SPLINE
SPL {X  -162.485, Y  +370.062, Z    +0.000, E1   +10.606, E3 +501495.136}
SPL {X  -162.818, Y  +379.636, Z    +0.000, E1    +5.115, E3 +501484.485}
SPL {X  -162.820, Y  +386.976, Z    +0.000, E1    +0.144, E3 +501483.584}
SPL {X  -162.820, Y  +390.236, Z    +0.000, E1    -2.204, E3 +501489.642}
SPL {X  -162.820, Y  +393.415, Z    +0.000, E1    -4.587, E3 +501490.927}
SPL {X  -162.820, Y  +399.630, Z    +0.000, E1    -9.426, E3 +501492.856}
SPL {X  -162.820, Y  +408.127, Z    +0.000, E1   -18.417, E3 +501479.144}
SPL {X  -162.820, Y  +420.083, Z    +0.000, E1   -24.325, E3 +501499.620}
SPL {X  -162.820, Y  +428.527, Z    +0.000, E1   -26.988, E3 +501516.912}
SPL {X  -162.820, Y  +431.336, Z    +0.000, E1   -24.162, E3 +501547.122}
SPL {X  -162.820, Y  +432.048, Z    +0.000, E1   -22.832, E3 +501561.626}
SPL {X  -162.820, Y  +434.888, Z    +0.000, E1   -22.823, E3 +501575.575}
SPL {X  -162.820, Y  +436.834, Z    +0.000, E1   -22.779, E3 +501585.535}
SPL {X  -162.820, Y  +438.868, Z    +0.000, E1   -22.837, E3 +501595.189}
SPL {X  -162.820, Y  +441.351, Z    +0.000, E1   -22.805, E3 +501607.764}
SPL {X  -162.820, Y  +443.809, Z    +0.000, E1   -22.804, E3 +501619.930}
SPL {X  -162.820, Y  +447.077, Z    +0.000, E1   -22.869, E3 +501635.741}
SPL {X  -162.820, Y  +449.911, Z    +0.000, E1   -22.774, E3 +501650.350}
SPL {X  -162.820, Y  +451.861, Z    +0.000, E1   -22.750, E3 +501660.198}
SPL {X  -162.820, Y  +454.167, Z    +0.000, E1   -22.842, E3 +501670.927}
SPL {X  -162.820, Y  +456.529, Z    +0.000, E1   -22.855, E3 +501682.456}
SPL {X  -162.820, Y  +458.725, Z    +0.000, E1   -22.793, E3 +501693.860}
SPL {X  -162.820, Y  +460.754, Z    +0.000, E1   -22.806, E3 +501703.733}
SPL {X  -162.820, Y  +462.409, Z    +0.000, E1   -22.783, E3 +501712.150}
SPL {X  -162.820, Y  +464.633, Z    +0.000, E1   -22.813, E3 +501722.979}
SPL {X  -162.820, Y  +467.913, Z    +0.000, E1   -22.879, E3 +501738.819}
SPL {X  -162.820, Y  +470.892, Z    +0.000, E1   -22.837, E3 +501753.708}
SPL {X  -162.820, Y  +472.726, Z    +0.000, E1   -22.777, E3 +501763.247}
SPL {X  -162.820, Y  +475.118, Z    +0.000, E1   -22.777, E3 +501775.218}
SPL {X  -162.820, Y  +477.389, Z    +0.000, E1   -22.803, E3 +501786.135}
SPL {X  -162.820, Y  +478.914, Z    +0.000, E1   -22.821, E3 +501793.526}
SPL {X  -162.820, Y  +481.034, Z    +0.000, E1   -22.831, E3 +501804.048}
SPL {X  -162.820, Y  +484.256, Z    +0.000, E1   -22.840, E3 +501820.067}
SPL {X  -162.820, Y  +487.952, Z    +0.000, E1   -22.824, E3 +501838.497}
SPL {X  -162.820, Y  +491.768, Z    +0.000, E1   -22.852, E3 +501857.178}
SPL {X  -162.820, Y  +495.526, Z    +0.000, E1   -22.833, E3 +501875.949}
SPL {X  -162.820, Y  +499.330, Z    +0.000, E1   -22.841, E3 +501894.730}
SPL {X  -162.820, Y  +503.049, Z    +0.000, E1   -22.823, E3 +501913.280}
SPL {X  -162.820, Y  +506.908, Z    +0.000, E1   -22.877, E3 +501931.950}
SPL {X  -162.820, Y  +510.068, Z    +0.000, E1   -22.761, E3 +501948.421}
SPL {X  -162.820, Y  +512.359, Z    +0.000, E1   -22.823, E3 +501959.153}
SPL {X  -162.820, Y  +514.562, Z    +0.000, E1   -22.806, E3 +501970.340}
SPL {X  -162.820, Y  +517.952, Z    +0.000, E1   -22.864, E3 +501986.737}
SPL {X  -162.820, Y  +520.641, Z    +0.000, E1   -22.790, E3 +502000.456}
SPL {X  -162.820, Y  +522.740, Z    +0.000, E1   -22.811, E3 +502010.698}
SPL {X  -162.820, Y  +524.628, Z    +0.000, E1   -22.846, E3 +502019.693}
SPL {X  -162.820, Y  +526.661, Z    +0.000, E1   -22.801, E3 +502030.249}
SPL {X  -162.820, Y  +529.662, Z    +0.000, E1   -22.810, E3 +502045.099}
SPL {X  -162.820, Y  +532.614, Z    +0.000, E1   -22.828, E3 +502059.506}
SPL {X  -162.820, Y  +534.838, Z    +0.000, E1   -22.864, E3 +502070.134}
SPL {X  -162.820, Y  +536.882, Z    +0.000, E1   -22.782, E3 +502080.989}
SPL {X  -162.820, Y  +539.194, Z    +0.000, E1   -22.826, E3 +502092.038}
SPL {X  -162.820, Y  +541.555, Z    +0.000, E1   -22.817, E3 +502103.852}
SPL {X  -162.820, Y  +543.728, Z    +0.000, E1   -22.799, E3 +502114.710}
SPL {X  -162.820, Y  +545.925, Z    +0.000, E1   -22.803, E3 +502125.580}
SPL {X  -162.820, Y  +548.328, Z    +0.000, E1   -22.796, E3 +502137.575}
SPL {X  -162.820, Y  +551.027, Z    +0.000, E1   -22.819, E3 +502150.768}
SPL {X  -162.820, Y  +553.721, Z    +0.000, E1   -22.807, E3 +502164.212}
SPL {X  -162.820, Y  +556.430, Z    +0.000, E1   -22.821, E3 +502177.508}
SPL {X  -162.820, Y  +558.974, Z    +0.000, E1   -22.806, E3 +502190.208}
SPL {X  -162.820, Y  +562.171, Z    +0.000, E1   -22.845, E3 +502205.906}
SPL {X  -162.820, Y  +565.170, Z    +0.000, E1   -22.801, E3 +502220.919}
SPL {X  -162.820, Y  +567.308, Z    +0.000, E1   -22.750, E3 +502231.936}
SPL {X  -162.820, Y  +570.378, Z    +0.000, E1   -22.843, E3 +502246.559}
SPL {X  -162.820, Y  +573.634, Z    +0.000, E1   -22.827, E3 +502262.703}
SPL {X  -162.820, Y  +576.228, Z    +0.000, E1   -22.814, E3 +502275.600}
SPL {X  -162.820, Y  +578.553, Z    +0.000, E1   -22.801, E3 +502287.215}
SPL {X  -162.820, Y  +581.064, Z    +0.000, E1   -22.823, E3 +502299.500}
SPL {X  -162.820, Y  +583.435, Z    +0.000, E1   -22.808, E3 +502311.322}
SPL {X  -162.820, Y  +585.410, Z    +0.000, E1   -22.764, E3 +502321.457}
SPL {X  -162.820, Y  +587.676, Z    +0.000, E1   -22.853, E3 +502331.972}
SPL {X  -162.820, Y  +590.707, Z    +0.000, E1   -22.855, E3 +502347.122}
SPL {X  -162.820, Y  +593.650, Z    +0.000, E1   -22.810, E3 +502361.882}
SPL {X  -162.820, Y  +595.830, Z    +0.000, E1   -22.828, E3 +502372.498}
SPL {X  -162.820, Y  +598.094, Z    +0.000, E1   -22.843, E3 +502383.611}
SPL {X  -162.820, Y  +600.420, Z    +0.000, E1   -22.826, E3 +502395.243}
SPL {X  -162.820, Y  +602.573, Z    +0.000, E1   -22.830, E3 +502405.828}
SPL {X  -162.820, Y  +604.828, Z    +0.000, E1   -22.784, E3 +502417.466}
SPL {X  -162.820, Y  +607.142, Z    +0.000, E1   -22.808, E3 +502428.647}
SPL {X  -162.820, Y  +608.890, Z    +0.000, E1   -22.790, E3 +502437.471}
SPL {X  -162.820, Y  +611.103, Z    +0.000, E1   -22.785, E3 +502448.510}
SPL {X  -162.820, Y  +613.294, Z    +0.000, E1   -22.780, E3 +502459.383}
SPL {X  -162.820, Y  +615.356, Z    +0.000, E1   -22.799, E3 +502469.440}
SPL {X  -162.820, Y  +617.439, Z    +0.000, E1   -22.808, E3 +502479.698}
SPL {X  -162.820, Y  +619.665, Z    +0.000, E1   -22.817, E3 +502490.666}
SPL {X  -162.820, Y  +621.733, Z    +0.000, E1   -22.759, E3 +502501.390}
SPL {X  -162.820, Y  +624.076, Z    +0.000, E1   -22.774, E3 +502512.896}
SPL {X  -162.820, Y  +627.244, Z    +0.000, E1   -22.803, E3 +502528.578}
SPL {X  -162.820, Y  +630.349, Z    +0.000, E1   -22.766, E3 +502544.110}
SPL {X  -162.820, Y  +632.572, Z    +0.000, E1   -22.785, E3 +502554.916}
SPL {X  -162.820, Y  +634.507, Z    +0.000, E1   -22.784, E3 +502564.555}
SPL {X  -162.820, Y  +636.863, Z    +0.000, E1   -22.760, E3 +502576.477}
SPL {X  -162.820, Y  +640.111, Z    +0.000, E1   -22.809, E3 +502592.360}
SPL {X  -162.820, Y  +643.449, Z    +0.000, E1   -22.796, E3 +502608.878}
SPL {X  -162.820, Y  +645.630, Z    +0.000, E1   -22.795, E3 +502619.574}
SPL {X  -162.820, Y  +647.561, Z    +0.000, E1   -22.705, E3 +502630.025}
SPL {X  -162.820, Y  +651.051, Z    +0.000, E1   -22.833, E3 +502646.444}
SPL {X  -162.820, Y  +653.898, Z    +0.000, E1   -22.796, E3 +502660.630}
SPL {X  -162.820, Y  +656.161, Z    +0.000, E1   -22.812, E3 +502671.751}
SPL {X  -162.820, Y  +658.384, Z    +0.000, E1   -22.822, E3 +502682.618}
SPL {X  -162.820, Y  +660.215, Z    +0.000, E1   -22.649, E3 +502693.208}
SPL {X  -162.820, Y  +662.823, Z    +0.000, E1   -22.799, E3 +502704.916}
SPL {X  -162.820, Y  +665.112, Z    +0.000, E1   -22.835, E3 +502715.971}
SPL {X  -162.820, Y  +667.016, Z    +0.000, E1   -22.823, E3 +502725.399}
SPL {X  -162.820, Y  +668.960, Z    +0.000, E1   -22.773, E3 +502735.566}
SPL {X  -162.820, Y  +671.605, Z    +0.000, E1   -22.777, E3 +502748.640}
SPL {X  -162.817, Y  +674.515, Z    +0.000, E1   -22.816, E3 +502762.837}
SPL {X  -162.773, Y  +677.428, Z    +0.000, E1   -22.762, E3 +502777.645}
SPL {X  -162.691, Y  +679.987, Z    +0.000, E1   -22.794, E3 +502790.058}
SPL {X  -162.559, Y  +682.717, Z    +0.000, E1   -22.726, E3 +502804.242}
SPL {X  -162.349, Y  +685.880, Z    +0.000, E1   -22.738, E3 +502819.843}
SPL {X  -162.090, Y  +688.902, Z    +0.000, E1   -22.700, E3 +502835.138}
SPL {X  -161.474, Y  +694.390, Z    +0.000, E1   -24.298, E3 +502848.493}
SPL {X  -158.553, Y  +710.529, Z    +0.000, E1   -30.890, E3 +502865.055}
ENDSPLINE

SPLINE
SPL {X  -161.215, Y  +696.305, Z    +0.000, E1   -20.575, E3 +502891.635}
SPL {X  -161.691, Y  +692.643, Z    +0.000, E1   -17.369, E3 +502907.824}
SPL {X  -162.534, Y  +683.153, Z    +0.000, E1   -10.475, E3 +502933.291}
SPL {X  -162.820, Y  +667.630, Z    +0.000, E1    -0.882, E3 +502927.267}
SPL {X  -162.820, Y  +661.883, Z    +0.000, E1    +3.373, E3 +502932.710}
SPL {X  -162.820, Y  +653.808, Z    +0.000, E1    +9.891, E3 +502930.402}
SPL {X  -162.820, Y  +632.548, Z    +0.000, E1   +27.446, E3 +502926.938}
ENDSPLINE

SPLINE
SPL {X  -162.820, Y  +638.080, Z    +0.000, E1   +18.858, E3 +502954.687}
ENDSPLINE

SPLINE
SPL {X  -162.820, Y  +623.278, Z    +0.000, E1   +28.723, E3 +502956.257}
SPL {X  -162.820, Y  +618.658, Z    +0.000, E1   +26.841, E3 +502984.866}
ENDSPLINE

SPLINE
SPL {X  -162.820, Y  +623.685, Z    +0.000, E1   +22.346, E3 +502997.173}
ENDSPLINE

SPLINE
SPL {X  -162.820, Y  +621.304, Z    +0.000, E1   +22.259, E3 +503009.988}
SPL {X  -162.820, Y  +618.758, Z    +0.000, E1   +22.239, E3 +503023.139}
SPL {X  -162.820, Y  +616.062, Z    +0.000, E1   +22.275, E3 +503036.560}
SPL {X  -162.820, Y  +613.536, Z    +0.000, E1   +22.242, E3 +503049.681}
SPL {X  -162.820, Y  +611.128, Z    +0.000, E1   +22.252, E3 +503061.852}
SPL {X  -162.820, Y  +608.428, Z    +0.000, E1   +22.255, E3 +503075.635}
SPL {X  -162.820, Y  +605.984, Z    +0.000, E1   +22.221, E3 +503088.272}
SPL {X  -162.820, Y  +603.020, Z    +0.000, E1   +22.272, E3 +503103.170}
SPL {X  -162.820, Y  +599.168, Z    +0.000, E1   +22.310, E3 +503122.438}
SPL {X  -162.820, Y  +596.569, Z    +0.000, E1   +22.222, E3 +503136.161}
SPL {X  -162.820, Y  +594.115, Z    +0.000, E1   +22.273, E3 +503148.386}
SPL {X  -162.820, Y  +591.721, Z    +0.000, E1   +22.239, E3 +503160.701}
SPL {X  -162.820, Y  +589.492, Z    +0.000, E1   +22.304, E3 +503171.562}
SPL {X  -162.820, Y  +587.447, Z    +0.000, E1   +22.279, E3 +503182.091}
SPL {X  -162.820, Y  +585.192, Z    +0.000, E1   +22.298, E3 +503193.501}
SPL {X  -162.820, Y  +582.610, Z    +0.000, E1   +22.234, E3 +503207.124}
SPL {X  -162.820, Y  +580.317, Z    +0.000, E1   +22.300, E3 +503218.178}
SPL {X  -162.820, Y  +578.878, Z    +0.000, E1   +22.272, E3 +503225.688}
SPL {X  -162.820, Y  +576.856, Z    +0.000, E1   +22.233, E3 +503236.446}
SPL {X  -162.820, Y  +573.830, Z    +0.000, E1   +22.272, E3 +503251.582}
SPL {X  -162.820, Y  +570.852, Z    +0.000, E1   +22.234, E3 +503267.042}
SPL {X  -162.820, Y  +568.608, Z    +0.000, E1   +22.253, E3 +503278.175}
SPL {X  -162.820, Y  +565.838, Z    +0.000, E1   +22.271, E3 +503292.406}
SPL {X  -162.820, Y  +562.162, Z    +0.000, E1   +22.252, E3 +503311.223}
SPL {X  -162.820, Y  +558.919, Z    +0.000, E1   +22.286, E3 +503327.387}
SPL {X  -162.820, Y  +555.548, Z    +0.000, E1   +22.322, E3 +503344.296}
SPL {X  -162.820, Y  +552.787, Z    +0.000, E1   +22.213, E3 +503359.093}
SPL {X  -162.820, Y  +550.136, Z    +0.000, E1   +22.258, E3 +503372.327}
SPL {X  -162.820, Y  +546.694, Z    +0.000, E1   +22.290, E3 +503389.649}
SPL {X  -162.820, Y  +543.558, Z    +0.000, E1   +22.285, E3 +503405.512}
SPL {X  -162.820, Y  +541.633, Z    +0.000, E1   +22.257, E3 +503415.440}
SPL {X  -162.820, Y  +539.116, Z    +0.000, E1   +22.302, E3 +503428.051}
SPL {X  -162.820, Y  +536.913, Z    +0.000, E1   +22.192, E3 +503439.975}
SPL {X  -162.820, Y  +534.880, Z    +0.000, E1   +22.252, E3 +503449.929}
SPL {X  -162.820, Y  +532.896, Z    +0.000, E1   +22.234, E3 +503460.089}
SPL {X  -162.820, Y  +531.056, Z    +0.000, E1   +22.251, E3 +503469.371}
SPL {X  -162.820, Y  +528.708, Z    +0.000, E1   +22.319, E3 +503480.752}
SPL {X  -162.820, Y  +525.932, Z    +0.000, E1   +22.258, E3 +503495.509}
SPL {X  -162.820, Y  +522.524, Z    +0.000, E1   +22.326, E3 +503512.233}
SPL {X  -162.820, Y  +519.457, Z    +0.000, E1   +22.481, E3 +503526.362}
SPL {X  -162.820, Y  +506.285, Z    +0.000, E1   +28.538, E3 +503537.819}
SPL {X  -162.820, Y  +504.441, Z    +0.000, E1   +27.574, E3 +503552.162}
SPL {X  -162.820, Y  +502.813, Z    +0.000, E1   +26.013, E3 +503570.359}
SPL {X  -162.820, Y  +502.016, Z    +0.000, E1   +24.802, E3 +503582.702}
SPL {X  -162.820, Y  +501.060, Z    +0.000, E1   +24.081, E3 +503592.891}
SPL {X  -162.820, Y  +499.934, Z    +0.000, E1   +22.814, E3 +503608.760}
SPL {X  -162.820, Y  +498.303, Z    +0.000, E1   +21.749, E3 +503626.016}
SPL {X  -162.820, Y  +495.897, Z    +0.000, E1   +21.662, E3 +503639.170}
SPL {X  -162.820, Y  +493.717, Z    +0.000, E1   +21.704, E3 +503650.276}
SPL {X  -162.820, Y  +491.396, Z    +0.000, E1   +21.707, E3 +503662.400}
SPL {X  -162.820, Y  +489.485, Z    +0.000, E1   +21.661, E3 +503672.748}
SPL {X  -162.820, Y  +487.723, Z    +0.000, E1   +21.665, E3 +503681.951}
SPL {X  -162.820, Y  +485.661, Z    +0.000, E1   +21.712, E3 +503692.395}
SPL {X  -162.820, Y  +482.775, Z    +0.000, E1   +21.716, E3 +503707.647}
SPL {X  -162.820, Y  +479.894, Z    +0.000, E1   +21.695, E3 +503722.723}
SPL {X  -162.820, Y  +477.685, Z    +0.000, E1   +21.656, E3 +503734.661}
SPL {X  -162.820, Y  +475.419, Z    +0.000, E1   +21.711, E3 +503746.014}
SPL {X  -162.820, Y  +473.301, Z    +0.000, E1   +21.712, E3 +503757.111}
SPL {X  -162.820, Y  +470.965, Z    +0.000, E1   +21.700, E3 +503769.456}
SPL {X  -162.820, Y  +469.036, Z    +0.000, E1   +21.695, E3 +503779.499}
SPL {X  -162.820, Y  +467.138, Z    +0.000, E1   +21.678, E3 +503789.671}
SPL {X  -162.820, Y  +465.011, Z    +0.000, E1   +21.692, E3 +503800.654}
SPL {X  -162.820, Y  +462.669, Z    +0.000, E1   +21.752, E3 +503812.434}
SPL {X  -162.820, Y  +460.725, Z    +0.000, E1   +21.689, E3 +503823.047}
SPL {X  -162.820, Y  +458.666, Z    +0.000, E1   +21.695, E3 +503833.859}
SPL {X  -162.820, Y  +456.431, Z    +0.000, E1   +21.708, E3 +503845.388}
SPL {X  -162.820, Y  +454.628, Z    +0.000, E1   +21.674, E3 +503855.106}
SPL {X  -162.820, Y  +452.690, Z    +0.000, E1   +21.773, E3 +503864.380}
SPL {X  -162.820, Y  +450.610, Z    +0.000, E1   +21.698, E3 +503875.979}
SPL {X  -162.820, Y  +448.170, Z    +0.000, E1   +21.667, E3 +503889.000}
SPL {X  -162.820, Y  +445.508, Z    +0.000, E1   +21.732, E3 +503902.518}
SPL {X  -162.820, Y  +442.443, Z    +0.000, E1   +21.712, E3 +503918.639}
SPL {X  -162.820, Y  +439.933, Z    +0.000, E1   +21.690, E3 +503931.919}
SPL {X  -162.820, Y  +437.628, Z    +0.000, E1   +21.678, E3 +503944.107}
SPL {X  -162.820, Y  +434.473, Z    +0.000, E1   +21.747, E3 +503960.204}
SPL {X  -162.820, Y  +431.492, Z    +0.000, E1   +21.686, E3 +503976.152}
SPL {X  -162.820, Y  +429.074, Z    +0.000, E1   +21.710, E3 +503988.604}
SPL {X  -162.820, Y  +426.023, Z    +0.000, E1   +21.718, E3 +504004.672}
SPL {X  -162.820, Y  +422.986, Z    +0.000, E1   +21.685, E3 +504020.720}
SPL {X  -162.820, Y  +420.528, Z    +0.000, E1   +21.706, E3 +504033.370}
SPL {X  -162.820, Y  +418.116, Z    +0.000, E1   +21.761, E3 +504045.517}
SPL {X  -162.820, Y  +416.127, Z    +0.000, E1   +21.715, E3 +504056.222}
SPL {X  -162.820, Y  +414.361, Z    +0.000, E1   +21.613, E3 +504066.409}
SPL {X  -162.820, Y  +411.450, Z    +0.000, E1   +21.710, E3 +504080.983}
SPL {X  -162.820, Y  +408.590, Z    +0.000, E1   +21.735, E3 +504095.608}
SPL {X  -162.820, Y  +406.238, Z    +0.000, E1   +21.697, E3 +504108.257}
SPL {X  -162.820, Y  +403.166, Z    +0.000, E1   +21.746, E3 +504124.063}
SPL {X  -162.820, Y  +400.348, Z    +0.000, E1   +21.713, E3 +504138.898}
SPL {X  -162.820, Y  +398.298, Z    +0.000, E1   +21.721, E3 +504149.514}
SPL {X  -162.820, Y  +396.371, Z    +0.000, E1   +21.713, E3 +504159.695}
SPL {X  -162.820, Y  +394.508, Z    +0.000, E1   +21.616, E3 +504170.251}
SPL {X  -162.820, Y  +391.777, Z    +0.000, E1   +21.714, E3 +504183.910}
SPL {X  -162.820, Y  +388.822, Z    +0.000, E1   +21.717, E3 +504199.230}
SPL {X  -162.820, Y  +386.818, Z    +0.000, E1   +21.679, E3 +504209.970}
SPL {X  -162.820, Y  +384.697, Z    +0.000, E1   +21.693, E3 +504221.040}
SPL {X  -162.820, Y  +382.288, Z    +0.000, E1   +21.742, E3 +504233.164}
SPL {X  -162.817, Y  +379.520, Z    +0.000, E1   +21.723, E3 +504248.001}
SPL {X  -162.776, Y  +376.710, Z    +0.000, E1   +21.698, E3 +504262.740}
SPL {X  -162.707, Y  +374.438, Z    +0.000, E1   +21.688, E3 +504274.744}
SPL {X  -162.607, Y  +372.171, Z    +0.000, E1   +21.692, E3 +504286.544}
SPL {X  -162.494, Y  +370.197, Z    +0.000, E1   +21.655, E3 +504297.170}
SPL {X  -162.349, Y  +368.131, Z    +0.000, E1   +21.624, E3 +504308.288}
SPL {X  -162.161, Y  +365.866, Z    +0.000, E1   +21.642, E3 +504319.973}
SPL {X  -161.651, Y  +361.024, Z    +0.000, E1   +22.970, E3 +504333.396}
SPL {X  -160.281, Y  +351.857, Z    +0.000, E1   +24.243, E3 +504368.735}
ENDSPLINE

SPLINE
SPL {X  -161.833, Y  +362.603, Z    +0.000, E1   +17.021, E3 +504383.431}
ENDSPLINE

SPLINE
SPL {X  -160.786, Y  +354.842, Z    +0.000, E1   +19.274, E3 +504415.587}
ENDSPLINE

SPLINE
SPL {X  -162.485, Y  +370.062, Z    +0.000, E1   +10.606, E3 +504421.965}
SPL {X  -162.818, Y  +379.636, Z    +0.000, E1    +5.115, E3 +504411.314}
SPL {X  -162.820, Y  +386.976, Z    +0.000, E1    +0.144, E3 +504410.413}
SPL {X  -162.820, Y  +390.236, Z    +0.000, E1    -2.204, E3 +504416.472}
SPL {X  -162.820, Y  +393.415, Z    +0.000, E1    -4.587, E3 +504417.756}
SPL {X  -162.820, Y  +399.630, Z    +0.000, E1    -9.426, E3 +504419.685}
SPL {X  -162.820, Y  +408.127, Z    +0.000, E1   -18.417, E3 +504405.974}
SPL {X  -162.820, Y  +420.083, Z    +0.000, E1   -24.325, E3 +504426.449}
SPL {X  -162.820, Y  +428.527, Z    +0.000, E1   -26.988, E3 +504443.741}
SPL {X  -162.820, Y  +431.191, Z    +0.000, E1   -23.548, E3 +504478.594}
SPL {X  -162.820, Y  +432.946, Z    +0.000, E1   -22.795, E3 +504492.998}
SPL {X  -162.820, Y  +434.888, Z    +0.000, E1   -22.823, E3 +504502.405}
SPL {X  -162.820, Y  +436.834, Z    +0.000, E1   -22.779, E3 +504512.365}
SPL {X  -162.820, Y  +438.868, Z    +0.000, E1   -22.837, E3 +504522.018}
SPL {X  -162.820, Y  +441.351, Z    +0.000, E1   -22.805, E3 +504534.594}
SPL {X  -162.820, Y  +443.809, Z    +0.000, E1   -22.804, E3 +504546.760}
SPL {X  -162.820, Y  +447.077, Z    +0.000, E1   -22.869, E3 +504562.570}
SPL {X  -162.820, Y  +449.911, Z    +0.000, E1   -22.774, E3 +504577.180}
SPL {X  -162.820, Y  +451.861, Z    +0.000, E1   -22.750, E3 +504587.027}
SPL {X  -162.820, Y  +454.167, Z    +0.000, E1   -22.842, E3 +504597.757}
SPL {X  -162.820, Y  +456.529, Z    +0.000, E1   -22.855, E3 +504609.285}
SPL {X  -162.820, Y  +458.725, Z    +0.000, E1   -22.793, E3 +504620.690}
SPL {X  -162.820, Y  +460.754, Z    +0.000, E1   -22.806, E3 +504630.563}
SPL {X  -162.820, Y  +462.409, Z    +0.000, E1   -22.783, E3 +504638.979}
SPL {X  -162.820, Y  +464.633, Z    +0.000, E1   -22.813, E3 +504649.809}
SPL {X  -162.820, Y  +467.913, Z    +0.000, E1   -22.879, E3 +504665.648}
SPL {X  -162.820, Y  +470.892, Z    +0.000, E1   -22.837, E3 +504680.537}
SPL {X  -162.820, Y  +472.726, Z    +0.000, E1   -22.777, E3 +504690.076}
SPL {X  -162.820, Y  +475.118, Z    +0.000, E1   -22.777, E3 +504702.047}
SPL {X  -162.820, Y  +477.389, Z    +0.000, E1   -22.803, E3 +504712.964}
SPL {X  -162.820, Y  +478.914, Z    +0.000, E1   -22.821, E3 +504720.356}
SPL {X  -162.820, Y  +481.034, Z    +0.000, E1   -22.831, E3 +504730.878}
SPL {X  -162.820, Y  +484.256, Z    +0.000, E1   -22.840, E3 +504746.896}
SPL {X  -162.820, Y  +487.952, Z    +0.000, E1   -22.824, E3 +504765.327}
SPL {X  -162.820, Y  +491.768, Z    +0.000, E1   -22.852, E3 +504784.007}
SPL {X  -162.820, Y  +495.526, Z    +0.000, E1   -22.833, E3 +504802.779}
SPL {X  -162.820, Y  +499.330, Z    +0.000, E1   -22.841, E3 +504821.560}
SPL {X  -162.820, Y  +503.049, Z    +0.000, E1   -22.823, E3 +504840.109}
SPL {X  -162.820, Y  +506.908, Z    +0.000, E1   -22.877, E3 +504858.779}
SPL {X  -162.820, Y  +510.068, Z    +0.000, E1   -22.761, E3 +504875.251}
SPL {X  -162.820, Y  +512.359, Z    +0.000, E1   -22.823, E3 +504885.982}
SPL {X  -162.820, Y  +513.873, Z    +0.000, E1   -22.800, E3 +504893.669}
SPL {X  -162.820, Y  +516.100, Z    +0.000, E1   -22.809, E3 +504904.745}
SPL {X  -162.820, Y  +518.662, Z    +0.000, E1   -22.847, E3 +504917.044}
SPL {X  -162.820, Y  +520.641, Z    +0.000, E1   -22.790, E3 +504927.285}
SPL {X  -162.820, Y  +523.535, Z    +0.000, E1   -22.857, E3 +504941.254}
SPL {X  -162.820, Y  +526.661, Z    +0.000, E1   -22.801, E3 +504957.078}
SPL {X  -162.820, Y  +528.725, Z    +0.000, E1   -22.770, E3 +504967.447}
SPL {X  -162.820, Y  +530.303, Z    +0.000, E1   -22.798, E3 +504975.066}
SPL {X  -162.820, Y  +532.614, Z    +0.000, E1   -22.828, E3 +504986.335}
SPL {X  -162.820, Y  +534.838, Z    +0.000, E1   -22.864, E3 +504996.964}
SPL {X  -162.820, Y  +536.882, Z    +0.000, E1   -22.782, E3 +505007.819}
SPL {X  -162.820, Y  +539.194, Z    +0.000, E1   -22.826, E3 +505018.867}
SPL {X  -162.820, Y  +541.555, Z    +0.000, E1   -22.817, E3 +505030.681}
SPL {X  -162.820, Y  +543.728, Z    +0.000, E1   -22.799, E3 +505041.539}
SPL {X  -162.820, Y  +545.925, Z    +0.000, E1   -22.803, E3 +505052.409}
SPL {X  -162.820, Y  +549.071, Z    +0.000, E1   -22.836, E3 +505067.936}
SPL {X  -162.820, Y  +553.089, Z    +0.000, E1   -22.838, E3 +505087.836}
SPL {X  -162.820, Y  +556.430, Z    +0.000, E1   -22.821, E3 +505104.337}
SPL {X  -162.820, Y  +558.974, Z    +0.000, E1   -22.806, E3 +505117.037}
SPL {X  -162.820, Y  +562.171, Z    +0.000, E1   -22.845, E3 +505132.735}
SPL {X  -162.820, Y  +565.170, Z    +0.000, E1   -22.801, E3 +505147.749}
SPL {X  -162.820, Y  +567.308, Z    +0.000, E1   -22.750, E3 +505158.765}
SPL {X  -162.820, Y  +570.378, Z    +0.000, E1   -22.843, E3 +505173.389}
SPL {X  -162.820, Y  +573.634, Z    +0.000, E1   -22.827, E3 +505189.533}
SPL {X  -162.820, Y  +576.228, Z    +0.000, E1   -22.814, E3 +505202.429}
SPL {X  -162.820, Y  +578.553, Z    +0.000, E1   -22.801, E3 +505214.045}
SPL {X  -162.820, Y  +581.064, Z    +0.000, E1   -22.823, E3 +505226.329}
SPL {X  -162.820, Y  +583.435, Z    +0.000, E1   -22.808, E3 +505238.151}
SPL {X  -162.820, Y  +585.410, Z    +0.000, E1   -22.764, E3 +505248.287}
SPL {X  -162.820, Y  +587.676, Z    +0.000, E1   -22.853, E3 +505258.801}
SPL {X  -162.820, Y  +590.707, Z    +0.000, E1   -22.855, E3 +505273.952}
SPL {X  -162.820, Y  +593.650, Z    +0.000, E1   -22.810, E3 +505288.712}
SPL {X  -162.820, Y  +595.830, Z    +0.000, E1   -22.828, E3 +505299.328}
SPL {X  -162.820, Y  +598.094, Z    +0.000, E1   -22.843, E3 +505310.441}
SPL {X  -162.820, Y  +600.420, Z    +0.000, E1   -22.826, E3 +505322.072}
SPL {X  -162.820, Y  +603.245, Z    +0.000, E1   -22.831, E3 +505336.137}
SPL {X  -162.820, Y  +606.456, Z    +0.000, E1   -22.811, E3 +505352.183}
SPL {X  -162.820, Y  +608.890, Z    +0.000, E1   -22.790, E3 +505364.301}
SPL {X  -162.820, Y  +611.103, Z    +0.000, E1   -22.785, E3 +505375.339}
SPL {X  -162.820, Y  +613.294, Z    +0.000, E1   -22.780, E3 +505386.212}
SPL {X  -162.820, Y  +615.356, Z    +0.000, E1   -22.799, E3 +505396.269}
SPL {X  -162.820, Y  +617.439, Z    +0.000, E1   -22.808, E3 +505406.527}
SPL {X  -162.820, Y  +619.665, Z    +0.000, E1   -22.817, E3 +505417.495}
SPL {X  -162.820, Y  +621.733, Z    +0.000, E1   -22.759, E3 +505428.220}
SPL {X  -162.820, Y  +624.076, Z    +0.000, E1   -22.774, E3 +505439.725}
SPL {X  -162.820, Y  +627.244, Z    +0.000, E1   -22.803, E3 +505455.407}
SPL {X  -162.820, Y  +630.349, Z    +0.000, E1   -22.766, E3 +505470.939}
SPL {X  -162.820, Y  +632.572, Z    +0.000, E1   -22.785, E3 +505481.746}
SPL {X  -162.820, Y  +634.507, Z    +0.000, E1   -22.784, E3 +505491.384}
SPL {X  -162.820, Y  +636.863, Z    +0.000, E1   -22.760, E3 +505503.307}
SPL {X  -162.820, Y  +640.111, Z    +0.000, E1   -22.809, E3 +505519.189}
SPL {X  -162.820, Y  +643.449, Z    +0.000, E1   -22.796, E3 +505535.707}
SPL {X  -162.820, Y  +645.630, Z    +0.000, E1   -22.795, E3 +505546.403}
SPL {X  -162.820, Y  +647.561, Z    +0.000, E1   -22.705, E3 +505556.854}
SPL {X  -162.820, Y  +649.758, Z    +0.000, E1   -22.780, E3 +505567.044}
SPL {X  -162.820, Y  +651.708, Z    +0.000, E1   -22.810, E3 +505576.538}
SPL {X  -162.820, Y  +653.898, Z    +0.000, E1   -22.796, E3 +505587.459}
SPL {X  -162.820, Y  +656.161, Z    +0.000, E1   -22.812, E3 +505598.581}
SPL {X  -162.820, Y  +658.384, Z    +0.000, E1   -22.822, E3 +505609.447}
SPL {X  -162.820, Y  +660.215, Z    +0.000, E1   -22.649, E3 +505620.038}
SPL {X  -162.820, Y  +662.823, Z    +0.000, E1   -22.799, E3 +505631.745}
SPL {X  -162.820, Y  +665.112, Z    +0.000, E1   -22.835, E3 +505642.800}
SPL {X  -162.820, Y  +667.016, Z    +0.000, E1   -22.823, E3 +505652.228}
SPL {X  -162.820, Y  +668.960, Z    +0.000, E1   -22.773, E3 +505662.396}
SPL {X  -162.820, Y  +671.605, Z    +0.000, E1   -22.777, E3 +505675.469}
SPL {X  -162.817, Y  +674.515, Z    +0.000, E1   -22.816, E3 +505689.666}
SPL {X  -162.773, Y  +677.428, Z    +0.000, E1   -22.762, E3 +505704.474}
SPL {X  -162.691, Y  +679.987, Z    +0.000, E1   -22.794, E3 +505716.888}
SPL {X  -162.604, Y  +681.880, Z    +0.000, E1   -22.691, E3 +505727.048}
SPL {X  -162.458, Y  +684.346, Z    +0.000, E1   -22.764, E3 +505738.842}
SPL {X  -162.229, Y  +687.364, Z    +0.000, E1   -22.685, E3 +505754.462}
SPL {X  -161.938, Y  +690.422, Z    +0.000, E1   -22.769, E3 +505768.868}
SPL {X  -161.065, Y  +697.344, Z    +0.000, E1   -25.698, E3 +505777.987}
SPL {X  -158.730, Y  +709.763, Z    +0.000, E1   -31.225, E3 +505786.661}
ENDSPLINE

SPLINE
SPL {X  -160.932, Y  +698.225, Z    +0.000, E1   -21.712, E3 +505817.770}
SPL {X  -161.917, Y  +690.622, Z    +0.000, E1   -16.445, E3 +505831.371}
ENDSPLINE

SPLINE
SPL {X  -161.349, Y  +695.340, Z    +0.000, E1   -18.625, E3 +505838.989}
ENDSPLINE

SPLINE
SPL {X  -162.534, Y  +683.153, Z    +0.000, E1   -10.475, E3 +505860.120}
SPL {X  -162.820, Y  +667.630, Z    +0.000, E1    -0.882, E3 +505854.096}
SPL {X  -162.820, Y  +661.883, Z    +0.000, E1    +3.373, E3 +505859.540}
SPL {X  -162.820, Y  +655.163, Z    +0.000, E1    +8.702, E3 +505859.138}
SPL {X  -162.820, Y  +634.515, Z    +0.000, E1   +26.439, E3 +505851.552}
ENDSPLINE

SPLINE
SPL {X  -162.820, Y  +638.080, Z    +0.000, E1   +18.858, E3 +505881.516}
ENDSPLINE

SPLINE
SPL {X  -162.820, Y  +623.278, Z    +0.000, E1   +28.723, E3 +505883.087}
SPL {X  -162.820, Y  +618.658, Z    +0.000, E1   +26.841, E3 +505911.696}
ENDSPLINE

SPLINE
SPL {X  -162.820, Y  +623.685, Z    +0.000, E1   +22.346, E3 +505924.002}
ENDSPLINE

SPLINE
SPL {X  -162.820, Y  +621.304, Z    +0.000, E1   +22.259, E3 +505936.817}
SPL {X  -162.820, Y  +618.758, Z    +0.000, E1   +22.239, E3 +505949.968}
SPL {X  -162.820, Y  +616.062, Z    +0.000, E1   +22.275, E3 +505963.389}
SPL {X  -162.820, Y  +613.536, Z    +0.000, E1   +22.242, E3 +505976.510}
SPL {X  -162.820, Y  +610.461, Z    +0.000, E1   +22.264, E3 +505992.142}
SPL {X  -162.820, Y  +607.796, Z    +0.000, E1   +22.261, E3 +506005.513}
SPL {X  -162.820, Y  +605.178, Z    +0.000, E1   +22.267, E3 +506018.997}
SPL {X  -162.820, Y  +602.350, Z    +0.000, E1   +22.224, E3 +506033.614}
SPL {X  -162.820, Y  +599.842, Z    +0.000, E1   +22.298, E3 +506045.765}
SPL {X  -162.820, Y  +597.194, Z    +0.000, E1   +22.253, E3 +506059.686}
SPL {X  -162.820, Y  +594.779, Z    +0.000, E1   +22.284, E3 +506071.590}
SPL {X  -162.820, Y  +592.389, Z    +0.000, E1   +22.245, E3 +506084.207}
SPL {X  -162.820, Y  +589.492, Z    +0.000, E1   +22.304, E3 +506098.391}
SPL {X  -162.820, Y  +587.447, Z    +0.000, E1   +22.279, E3 +506108.920}
SPL {X  -162.820, Y  +585.192, Z    +0.000, E1   +22.298, E3 +506120.330}
SPL {X  -162.820, Y  +582.610, Z    +0.000, E1   +22.234, E3 +506133.954}
SPL {X  -162.820, Y  +579.691, Z    +0.000, E1   +22.312, E3 +506148.225}
SPL {X  -162.820, Y  +577.460, Z    +0.000, E1   +22.218, E3 +506160.212}
SPL {X  -162.820, Y  +575.394, Z    +0.000, E1   +22.240, E3 +506170.637}
SPL {X  -162.820, Y  +572.645, Z    +0.000, E1   +22.246, E3 +506184.635}
SPL {X  -162.820, Y  +570.282, Z    +0.000, E1   +22.231, E3 +506196.685}
SPL {X  -162.820, Y  +567.961, Z    +0.000, E1   +22.247, E3 +506208.475}
SPL {X  -162.820, Y  +564.506, Z    +0.000, E1   +22.298, E3 +506225.789}
SPL {X  -162.820, Y  +561.620, Z    +0.000, E1   +22.191, E3 +506241.170}
SPL {X  -162.820, Y  +559.515, Z    +0.000, E1   +22.273, E3 +506251.171}
SPL {X  -162.820, Y  +556.723, Z    +0.000, E1   +22.309, E3 +506265.255}
SPL {X  -162.820, Y  +553.294, Z    +0.000, E1   +22.266, E3 +506283.043}
SPL {X  -162.820, Y  +550.871, Z    +0.000, E1   +22.229, E3 +506295.517}
SPL {X  -162.820, Y  +548.168, Z    +0.000, E1   +22.298, E3 +506308.853}
SPL {X  -162.820, Y  +545.860, Z    +0.000, E1   +22.216, E3 +506321.111}
SPL {X  -162.820, Y  +543.558, Z    +0.000, E1   +22.285, E3 +506332.341}
SPL {X  -162.820, Y  +540.968, Z    +0.000, E1   +22.274, E3 +506345.614}
SPL {X  -162.820, Y  +538.512, Z    +0.000, E1   +22.287, E3 +506357.926}
SPL {X  -162.820, Y  +535.523, Z    +0.000, E1   +22.266, E3 +506373.542}
SPL {X  -162.820, Y  +531.757, Z    +0.000, E1   +22.276, E3 +506392.596}
SPL {X  -162.820, Y  +527.980, Z    +0.000, E1   +22.326, E3 +506411.427}
SPL {X  -162.820, Y  +524.599, Z    +0.000, E1   +22.287, E3 +506428.824}
SPL {X  -162.820, Y  +522.011, Z    +0.000, E1   +22.282, E3 +506441.901}
SPL {X  -162.820, Y  +519.457, Z    +0.000, E1   +22.481, E3 +506453.191}
SPL {X  -162.820, Y  +505.859, Z    +0.000, E1   +28.367, E3 +506467.674}
SPL {X  -162.820, Y  +504.131, Z    +0.000, E1   +27.325, E3 +506481.812}
SPL {X  -162.820, Y  +503.215, Z    +0.000, E1   +26.369, E3 +506492.498}
SPL {X  -162.820, Y  +502.502, Z    +0.000, E1   +25.597, E3 +506501.345}
SPL {X  -162.820, Y  +501.672, Z    +0.000, E1   +24.583, E3 +506512.960}
SPL {X  -162.820, Y  +500.515, Z    +0.000, E1   +23.444, E3 +506527.490}
SPL {X  -162.820, Y  +499.633, Z    +0.000, E1   +22.486, E3 +506539.536}
SPL {X  -162.820, Y  +498.303, Z    +0.000, E1   +21.749, E3 +506552.845}
SPL {X  -162.820, Y  +495.897, Z    +0.000, E1   +21.662, E3 +506565.999}
SPL {X  -162.820, Y  +493.717, Z    +0.000, E1   +21.704, E3 +506577.105}
SPL {X  -162.820, Y  +491.396, Z    +0.000, E1   +21.707, E3 +506589.229}
SPL {X  -162.820, Y  +489.485, Z    +0.000, E1   +21.661, E3 +506599.577}
SPL {X  -162.820, Y  +487.723, Z    +0.000, E1   +21.665, E3 +506608.781}
SPL {X  -162.820, Y  +485.661, Z    +0.000, E1   +21.712, E3 +506619.224}
SPL {X  -162.820, Y  +482.775, Z    +0.000, E1   +21.716, E3 +506634.477}
SPL {X  -162.820, Y  +479.894, Z    +0.000, E1   +21.695, E3 +506649.553}
SPL {X  -162.820, Y  +477.685, Z    +0.000, E1   +21.656, E3 +506661.490}
SPL {X  -162.820, Y  +475.419, Z    +0.000, E1   +21.711, E3 +506672.843}
SPL {X  -162.820, Y  +473.301, Z    +0.000, E1   +21.712, E3 +506683.940}
SPL {X  -162.820, Y  +470.965, Z    +0.000, E1   +21.700, E3 +506696.285}
SPL {X  -162.820, Y  +469.036, Z    +0.000, E1   +21.695, E3 +506706.329}
SPL {X  -162.820, Y  +467.138, Z    +0.000, E1   +21.678, E3 +506716.500}
SPL {X  -162.820, Y  +465.011, Z    +0.000, E1   +21.692, E3 +506727.483}
SPL {X  -162.820, Y  +462.669, Z    +0.000, E1   +21.752, E3 +506739.263}
SPL {X  -162.820, Y  +460.725, Z    +0.000, E1   +21.689, E3 +506749.876}
SPL {X  -162.820, Y  +458.666, Z    +0.000, E1   +21.695, E3 +506760.688}
SPL {X  -162.820, Y  +456.431, Z    +0.000, E1   +21.708, E3 +506772.217}
SPL {X  -162.820, Y  +453.609, Z    +0.000, E1   +21.757, E3 +506786.751}
SPL {X  -162.820, Y  +450.610, Z    +0.000, E1   +21.698, E3 +506802.808}
SPL {X  -162.820, Y  +448.170, Z    +0.000, E1   +21.667, E3 +506815.829}
SPL {X  -162.820, Y  +445.508, Z    +0.000, E1   +21.732, E3 +506829.347}
SPL {X  -162.820, Y  +442.443, Z    +0.000, E1   +21.712, E3 +506845.468}
SPL {X  -162.820, Y  +439.933, Z    +0.000, E1   +21.690, E3 +506858.749}
SPL {X  -162.820, Y  +437.628, Z    +0.000, E1   +21.678, E3 +506870.937}
SPL {X  -162.820, Y  +434.473, Z    +0.000, E1   +21.747, E3 +506887.033}
SPL {X  -162.820, Y  +431.492, Z    +0.000, E1   +21.686, E3 +506902.982}
SPL {X  -162.820, Y  +429.074, Z    +0.000, E1   +21.710, E3 +506915.434}
SPL {X  -162.820, Y  +426.023, Z    +0.000, E1   +21.718, E3 +506931.501}
SPL {X  -162.820, Y  +422.986, Z    +0.000, E1   +21.685, E3 +506947.549}
SPL {X  -162.820, Y  +420.528, Z    +0.000, E1   +21.706, E3 +506960.199}
SPL {X  -162.820, Y  +418.116, Z    +0.000, E1   +21.761, E3 +506972.346}
SPL {X  -162.820, Y  +416.127, Z    +0.000, E1   +21.715, E3 +506983.051}
SPL {X  -162.820, Y  +414.361, Z    +0.000, E1   +21.613, E3 +506993.239}
SPL {X  -162.820, Y  +411.450, Z    +0.000, E1   +21.710, E3 +507007.812}
SPL {X  -162.820, Y  +408.590, Z    +0.000, E1   +21.735, E3 +507022.438}
SPL {X  -162.820, Y  +406.238, Z    +0.000, E1   +21.697, E3 +507035.087}
SPL {X  -162.820, Y  +403.166, Z    +0.000, E1   +21.746, E3 +507050.892}
SPL {X  -162.820, Y  +400.348, Z    +0.000, E1   +21.713, E3 +507065.727}
SPL {X  -162.820, Y  +398.298, Z    +0.000, E1   +21.721, E3 +507076.343}
SPL {X  -162.820, Y  +396.371, Z    +0.000, E1   +21.713, E3 +507086.525}
SPL {X  -162.820, Y  +394.508, Z    +0.000, E1   +21.616, E3 +507097.080}
SPL {X  -162.820, Y  +391.777, Z    +0.000, E1   +21.714, E3 +507110.739}
SPL {X  -162.820, Y  +388.822, Z    +0.000, E1   +21.717, E3 +507126.059}
SPL {X  -162.820, Y  +386.818, Z    +0.000, E1   +21.679, E3 +507136.799}
SPL {X  -162.820, Y  +384.697, Z    +0.000, E1   +21.693, E3 +507147.869}
SPL {X  -162.820, Y  +382.288, Z    +0.000, E1   +21.742, E3 +507159.993}
SPL {X  -162.817, Y  +379.520, Z    +0.000, E1   +21.723, E3 +507174.830}
SPL {X  -162.776, Y  +376.710, Z    +0.000, E1   +21.698, E3 +507189.569}
SPL {X  -162.707, Y  +374.438, Z    +0.000, E1   +21.688, E3 +507201.573}
SPL {X  -162.607, Y  +372.171, Z    +0.000, E1   +21.692, E3 +507213.373}
SPL {X  -162.494, Y  +370.197, Z    +0.000, E1   +21.655, E3 +507223.999}
SPL {X  -162.349, Y  +368.131, Z    +0.000, E1   +21.624, E3 +507235.117}
SPL {X  -162.161, Y  +365.866, Z    +0.000, E1   +21.642, E3 +507246.802}
SPL {X  -161.927, Y  +363.466, Z    +0.000, E1   +21.730, E3 +507258.574}
SPL {X  -160.290, Y  +351.907, Z    +0.000, E1   +27.562, E3 +507266.152}
SPL {X  -159.725, Y  +348.905, Z    +0.000, E1   +26.136, E3 +507291.387}
ENDSPLINE

SPLINE
SPL {X  -160.871, Y  +355.385, Z    +0.000, E1   +21.841, E3 +507300.230}
SPL {X  -161.833, Y  +362.603, Z    +0.000, E1   +17.021, E3 +507310.261}
ENDSPLINE

SPLINE
SPL {X  -160.786, Y  +354.842, Z    +0.000, E1   +19.274, E3 +507342.416}
ENDSPLINE

SPLINE
SPL {X  -162.485, Y  +370.062, Z    +0.000, E1   +10.606, E3 +507348.794}
SPL {X  -162.820, Y  +381.311, Z    +0.000, E1    +4.054, E3 +507339.150}
SPL {X  -162.820, Y  +389.994, Z    +0.000, E1    -2.149, E3 +507333.562}
SPL {X  -162.820, Y  +391.982, Z    +0.000, E1    -3.443, E3 +507344.007}
SPL {X  -162.820, Y  +399.630, Z    +0.000, E1    -9.426, E3 +507346.515}
SPL {X  -162.820, Y  +408.127, Z    +0.000, E1   -18.417, E3 +507332.803}
SPL {X  -162.820, Y  +420.083, Z    +0.000, E1   -24.325, E3 +507353.279}
SPL {X  -162.820, Y  +428.527, Z    +0.000, E1   -26.988, E3 +507370.571}
SPL {X  -162.820, Y  +431.191, Z    +0.000, E1   -23.548, E3 +507405.424}
SPL {X  -162.820, Y  +432.946, Z    +0.000, E1   -22.795, E3 +507419.827}
SPL {X  -162.820, Y  +434.888, Z    +0.000, E1   -22.823, E3 +507429.234}
SPL {X  -162.820, Y  +436.834, Z    +0.000, E1   -22.779, E3 +507439.194}
SPL {X  -162.820, Y  +438.868, Z    +0.000, E1   -22.837, E3 +507448.847}
SPL {X  -162.820, Y  +441.351, Z    +0.000, E1   -22.805, E3 +507461.423}
SPL {X  -162.820, Y  +443.809, Z    +0.000, E1   -22.804, E3 +507473.589}
SPL {X  -162.820, Y  +447.077, Z    +0.000, E1   -22.869, E3 +507489.399}
SPL {X  -162.820, Y  +449.911, Z    +0.000, E1   -22.774, E3 +507504.009}
SPL {X  -162.820, Y  +451.861, Z    +0.000, E1   -22.750, E3 +507513.856}
SPL {X  -162.820, Y  +454.167, Z    +0.000, E1   -22.842, E3 +507524.586}
SPL {X  -162.820, Y  +456.529, Z    +0.000, E1   -22.855, E3 +507536.114}
SPL {X  -162.820, Y  +458.725, Z    +0.000, E1   -22.793, E3 +507547.519}
SPL {X  -162.820, Y  +460.754, Z    +0.000, E1   -22.806, E3 +507557.392}
SPL {X  -162.820, Y  +462.409, Z    +0.000, E1   -22.783, E3 +507565.808}
SPL {X  -162.820, Y  +464.633, Z    +0.000, E1   -22.813, E3 +507576.638}
SPL {X  -162.820, Y  +467.913, Z    +0.000, E1   -22.879, E3 +507592.477}
SPL {X  -162.820, Y  +470.892, Z    +0.000, E1   -22.837, E3 +507607.366}
SPL {X  -162.820, Y  +472.726, Z    +0.000, E1   -22.777, E3 +507616.905}
SPL {X  -162.820, Y  +475.118, Z    +0.000, E1   -22.777, E3 +507628.877}
SPL {X  -162.820, Y  +477.389, Z    +0.000, E1   -22.803, E3 +507639.793}
SPL {X  -162.820, Y  +478.914, Z    +0.000, E1   -22.821, E3 +507647.185}
SPL {X  -162.820, Y  +481.034, Z    +0.000, E1   -22.831, E3 +507657.707}
SPL {X  -162.820, Y  +484.256, Z    +0.000, E1   -22.840, E3 +507673.726}
SPL {X  -162.820, Y  +487.952, Z    +0.000, E1   -22.824, E3 +507692.156}
SPL {X  -162.820, Y  +491.768, Z    +0.000, E1   -22.852, E3 +507710.837}
SPL {X  -162.820, Y  +495.526, Z    +0.000, E1   -22.833, E3 +507729.608}
SPL {X  -162.820, Y  +499.330, Z    +0.000, E1   -22.841, E3 +507748.389}
SPL {X  -162.820, Y  +503.049, Z    +0.000, E1   -22.823, E3 +507766.938}
SPL {X  -162.820, Y  +506.908, Z    +0.000, E1   -22.877, E3 +507785.608}
SPL {X  -162.820, Y  +510.068, Z    +0.000, E1   -22.761, E3 +507802.080}
SPL {X  -162.820, Y  +512.359, Z    +0.000, E1   -22.823, E3 +507812.811}
SPL {X  -162.820, Y  +513.873, Z    +0.000, E1   -22.800, E3 +507820.498}
SPL {X  -162.820, Y  +516.100, Z    +0.000, E1   -22.809, E3 +507831.575}
SPL {X  -162.820, Y  +518.662, Z    +0.000, E1   -22.847, E3 +507843.873}
SPL {X  -162.820, Y  +520.641, Z    +0.000, E1   -22.790, E3 +507854.114}
SPL {X  -162.820, Y  +523.535, Z    +0.000, E1   -22.857, E3 +507868.083}
SPL {X  -162.820, Y  +526.661, Z    +0.000, E1   -22.801, E3 +507883.907}
SPL {X  -162.820, Y  +528.725, Z    +0.000, E1   -22.770, E3 +507894.276}
SPL {X  -162.820, Y  +530.303, Z    +0.000, E1   -22.798, E3 +507901.896}
SPL {X  -162.820, Y  +532.614, Z    +0.000, E1   -22.828, E3 +507913.164}
SPL {X  -162.820, Y  +534.838, Z    +0.000, E1   -22.864, E3 +507923.793}
SPL {X  -162.820, Y  +536.882, Z    +0.000, E1   -22.782, E3 +507934.648}
SPL {X  -162.820, Y  +539.194, Z    +0.000, E1   -22.826, E3 +507945.696}
SPL {X  -162.820, Y  +541.555, Z    +0.000, E1   -22.817, E3 +507957.511}
SPL {X  -162.820, Y  +543.728, Z    +0.000, E1   -22.799, E3 +507968.368}
SPL {X  -162.820, Y  +545.925, Z    +0.000, E1   -22.803, E3 +507979.238}
SPL {X  -162.820, Y  +548.328, Z    +0.000, E1   -22.796, E3 +507991.234}
SPL {X  -162.820, Y  +551.027, Z    +0.000, E1   -22.819, E3 +508004.427}
SPL {X  -162.820, Y  +553.721, Z    +0.000, E1   -22.807, E3 +508017.871}
SPL {X  -162.820, Y  +556.430, Z    +0.000, E1   -22.821, E3 +508031.167}
SPL {X  -162.820, Y  +559.675, Z    +0.000, E1   -22.837, E3 +508047.247}
SPL {X  -162.820, Y  +562.799, Z    +0.000, E1   -22.814, E3 +508062.753}
SPL {X  -162.820, Y  +565.170, Z    +0.000, E1   -22.801, E3 +508074.578}
SPL {X  -162.820, Y  +568.020, Z    +0.000, E1   -22.787, E3 +508088.965}
SPL {X  -162.820, Y  +570.992, Z    +0.000, E1   -22.834, E3 +508103.184}
SPL {X  -162.820, Y  +572.901, Z    +0.000, E1   -22.775, E3 +508113.052}
SPL {X  -162.820, Y  +575.638, Z    +0.000, E1   -22.855, E3 +508126.162}
SPL {X  -162.820, Y  +578.553, Z    +0.000, E1   -22.801, E3 +508140.874}
SPL {X  -162.820, Y  +581.064, Z    +0.000, E1   -22.823, E3 +508153.158}
SPL {X  -162.820, Y  +583.435, Z    +0.000, E1   -22.808, E3 +508164.980}
SPL {X  -162.820, Y  +585.410, Z    +0.000, E1   -22.764, E3 +508175.116}
SPL {X  -162.820, Y  +587.676, Z    +0.000, E1   -22.853, E3 +508185.630}
SPL {X  -162.820, Y  +589.682, Z    +0.000, E1   -22.776, E3 +508196.160}
SPL {X  -162.820, Y  +591.720, Z    +0.000, E1   -22.868, E3 +508205.471}
SPL {X  -162.820, Y  +593.650, Z    +0.000, E1   -22.810, E3 +508215.541}
SPL {X  -162.820, Y  +595.830, Z    +0.000, E1   -22.828, E3 +508226.157}
SPL {X  -162.820, Y  +598.094, Z    +0.000, E1   -22.843, E3 +508237.270}
SPL {X  -162.820, Y  +600.420, Z    +0.000, E1   -22.826, E3 +508248.901}
SPL {X  -162.820, Y  +602.573, Z    +0.000, E1   -22.830, E3 +508259.486}
SPL {X  -162.820, Y  +604.828, Z    +0.000, E1   -22.784, E3 +508271.125}
SPL {X  -162.820, Y  +608.133, Z    +0.000, E1   -22.831, E3 +508287.243}
SPL {X  -162.820, Y  +611.103, Z    +0.000, E1   -22.785, E3 +508302.168}
SPL {X  -162.820, Y  +613.294, Z    +0.000, E1   -22.780, E3 +508313.041}
SPL {X  -162.820, Y  +615.356, Z    +0.000, E1   -22.799, E3 +508323.099}
SPL {X  -162.820, Y  +617.439, Z    +0.000, E1   -22.808, E3 +508333.357}
SPL {X  -162.820, Y  +619.665, Z    +0.000, E1   -22.817, E3 +508344.325}
SPL {X  -162.820, Y  +621.733, Z    +0.000, E1   -22.759, E3 +508355.049}
SPL {X  -162.820, Y  +624.076, Z    +0.000, E1   -22.774, E3 +508366.554}
SPL {X  -162.820, Y  +627.244, Z    +0.000, E1   -22.803, E3 +508382.236}
SPL {X  -162.820, Y  +630.349, Z    +0.000, E1   -22.766, E3 +508397.768}
SPL {X  -162.820, Y  +632.572, Z    +0.000, E1   -22.785, E3 +508408.575}
SPL {X  -162.820, Y  +634.507, Z    +0.000, E1   -22.784, E3 +508418.214}
SPL {X  -162.820, Y  +636.863, Z    +0.000, E1   -22.760, E3 +508430.136}
SPL {X  -162.820, Y  +640.111, Z    +0.000, E1   -22.809, E3 +508446.019}
SPL {X  -162.820, Y  +643.449, Z    +0.000, E1   -22.796, E3 +508462.536}
SPL {X  -162.820, Y  +645.630, Z    +0.000, E1   -22.795, E3 +508473.232}
SPL {X  -162.820, Y  +647.561, Z    +0.000, E1   -22.705, E3 +508483.683}
SPL {X  -162.820, Y  +649.758, Z    +0.000, E1   -22.780, E3 +508493.873}
SPL {X  -162.820, Y  +651.708, Z    +0.000, E1   -22.810, E3 +508503.368}
SPL {X  -162.820, Y  +653.898, Z    +0.000, E1   -22.796, E3 +508514.288}
SPL {X  -162.820, Y  +656.161, Z    +0.000, E1   -22.812, E3 +508525.410}
SPL {X  -162.820, Y  +658.384, Z    +0.000, E1   -22.822, E3 +508536.276}
SPL {X  -162.820, Y  +660.215, Z    +0.000, E1   -22.649, E3 +508546.867}
SPL {X  -162.820, Y  +662.823, Z    +0.000, E1   -22.799, E3 +508558.575}
SPL {X  -162.820, Y  +665.112, Z    +0.000, E1   -22.835, E3 +508569.629}
SPL {X  -162.820, Y  +667.016, Z    +0.000, E1   -22.823, E3 +508579.057}
SPL {X  -162.820, Y  +668.960, Z    +0.000, E1   -22.773, E3 +508589.225}
SPL {X  -162.820, Y  +672.333, Z    +0.000, E1   -22.837, E3 +508605.561}
SPL {X  -162.812, Y  +675.071, Z    +0.000, E1   -22.742, E3 +508619.706}
SPL {X  -162.773, Y  +677.428, Z    +0.000, E1   -22.762, E3 +508631.304}
SPL {X  -162.691, Y  +679.987, Z    +0.000, E1   -22.794, E3 +508643.717}
SPL {X  -162.604, Y  +681.880, Z    +0.000, E1   -22.691, E3 +508653.878}
SPL {X  -162.458, Y  +684.346, Z    +0.000, E1   -22.764, E3 +508665.671}
SPL {X  -162.296, Y  +686.547, Z    +0.000, E1   -22.660, E3 +508677.288}
SPL {X  -162.090, Y  +688.902, Z    +0.000, E1   -22.700, E3 +508688.796}
SPL {X  -161.474, Y  +694.390, Z    +0.000, E1   -24.298, E3 +508702.151}
SPL {X  -158.553, Y  +710.529, Z    +0.000, E1   -30.890, E3 +508718.713}
ENDSPLINE

SPLINE
SPL {X  -161.215, Y  +696.305, Z    +0.000, E1   -20.575, E3 +508745.294}
SPL {X  -161.691, Y  +692.643, Z    +0.000, E1   -17.369, E3 +508761.482}
SPL {X  -162.534, Y  +683.153, Z    +0.000, E1   -10.475, E3 +508786.949}
SPL {X  -162.820, Y  +667.630, Z    +0.000, E1    -0.882, E3 +508780.926}
SPL {X  -162.820, Y  +661.883, Z    +0.000, E1    +3.373, E3 +508786.369}
SPL {X  -162.820, Y  +653.808, Z    +0.000, E1    +9.891, E3 +508784.060}
SPL {X  -162.820, Y  +632.548, Z    +0.000, E1   +27.446, E3 +508780.597}
ENDSPLINE

SPLINE
SPL {X  -162.820, Y  +638.080, Z    +0.000, E1   +18.858, E3 +508808.345}
ENDSPLINE

SPLINE
SPL {X  -162.820, Y  +623.278, Z    +0.000, E1   +28.723, E3 +508809.916}
SPL {X  -162.820, Y  +618.658, Z    +0.000, E1   +26.841, E3 +508838.525}
ENDSPLINE

SPLINE
SPL {X  -162.820, Y  +623.685, Z    +0.000, E1   +22.346, E3 +508850.832}
ENDSPLINE

SPLINE
SPL {X  -162.820, Y  +621.304, Z    +0.000, E1   +22.259, E3 +508863.647}
SPL {X  -162.820, Y  +618.758, Z    +0.000, E1   +22.239, E3 +508876.798}
SPL {X  -162.820, Y  +616.062, Z    +0.000, E1   +22.275, E3 +508890.218}
SPL {X  -162.820, Y  +613.536, Z    +0.000, E1   +22.242, E3 +508903.340}
SPL {X  -162.820, Y  +611.128, Z    +0.000, E1   +22.252, E3 +508915.510}
SPL {X  -162.820, Y  +608.428, Z    +0.000, E1   +22.255, E3 +508929.294}
SPL {X  -162.820, Y  +605.178, Z    +0.000, E1   +22.267, E3 +508945.826}
SPL {X  -162.820, Y  +602.350, Z    +0.000, E1   +22.224, E3 +508960.443}
SPL {X  -162.820, Y  +599.842, Z    +0.000, E1   +22.298, E3 +508972.595}
SPL {X  -162.820, Y  +597.194, Z    +0.000, E1   +22.253, E3 +508986.516}
SPL {X  -162.820, Y  +594.779, Z    +0.000, E1   +22.284, E3 +508998.420}
SPL {X  -162.820, Y  +592.389, Z    +0.000, E1   +22.245, E3 +509011.036}
SPL {X  -162.820, Y  +589.492, Z    +0.000, E1   +22.304, E3 +509025.220}
SPL {X  -162.820, Y  +586.660, Z    +0.000, E1   +22.307, E3 +509039.661}
SPL {X  -162.820, Y  +583.204, Z    +0.000, E1   +22.278, E3 +509057.566}
SPL {X  -162.820, Y  +580.317, Z    +0.000, E1   +22.300, E3 +509071.837}
SPL {X  -162.820, Y  +578.061, Z    +0.000, E1   +22.264, E3 +509083.722}
SPL {X  -162.820, Y  +575.394, Z    +0.000, E1   +22.240, E3 +509097.466}
SPL {X  -162.820, Y  +573.156, Z    +0.000, E1   +22.254, E3 +509108.676}
SPL {X  -162.820, Y  +570.852, Z    +0.000, E1   +22.234, E3 +509120.700}
SPL {X  -162.820, Y  +567.961, Z    +0.000, E1   +22.247, E3 +509135.304}
SPL {X  -162.820, Y  +564.506, Z    +0.000, E1   +22.298, E3 +509152.618}
SPL {X  -162.820, Y  +561.620, Z    +0.000, E1   +22.191, E3 +509167.999}
SPL {X  -162.820, Y  +559.515, Z    +0.000, E1   +22.273, E3 +509178.001}
SPL {X  -162.820, Y  +556.723, Z    +0.000, E1   +22.309, E3 +509192.084}
SPL {X  -162.820, Y  +554.378, Z    +0.000, E1   +22.288, E3 +509203.930}
SPL {X  -162.820, Y  +552.787, Z    +0.000, E1   +22.213, E3 +509212.752}
SPL {X  -162.820, Y  +550.871, Z    +0.000, E1   +22.229, E3 +509222.346}
SPL {X  -162.820, Y  +548.168, Z    +0.000, E1   +22.298, E3 +509235.682}
SPL {X  -162.820, Y  +545.860, Z    +0.000, E1   +22.216, E3 +509247.940}
SPL {X  -162.820, Y  +543.558, Z    +0.000, E1   +22.285, E3 +509259.170}
SPL {X  -162.820, Y  +541.633, Z    +0.000, E1   +22.257, E3 +509269.099}
SPL {X  -162.820, Y  +539.116, Z    +0.000, E1   +22.302, E3 +509281.709}
SPL {X  -162.820, Y  +535.523, Z    +0.000, E1   +22.266, E3 +509300.371}
SPL {X  -162.820, Y  +531.757, Z    +0.000, E1   +22.276, E3 +509319.425}
SPL {X  -162.820, Y  +527.980, Z    +0.000, E1   +22.326, E3 +509338.256}
SPL {X  -162.820, Y  +524.599, Z    +0.000, E1   +22.287, E3 +509355.654}
SPL {X  -162.820, Y  +522.011, Z    +0.000, E1   +22.282, E3 +509368.731}
SPL {X  -162.820, Y  +519.457, Z    +0.000, E1   +22.481, E3 +509380.020}
SPL {X  -162.820, Y  +506.285, Z    +0.000, E1   +28.538, E3 +509391.478}
SPL {X  -162.820, Y  +504.441, Z    +0.000, E1   +27.574, E3 +509405.820}
SPL {X  -162.820, Y  +502.813, Z    +0.000, E1   +26.013, E3 +509424.018}
SPL {X  -162.820, Y  +502.016, Z    +0.000, E1   +24.802, E3 +509436.360}
SPL {X  -162.820, Y  +501.060, Z    +0.000, E1   +24.081, E3 +509446.550}
SPL {X  -162.820, Y  +500.336, Z    +0.000, E1   +23.110, E3 +509457.690}
SPL {X  -162.820, Y  +499.240, Z    +0.000, E1   +22.316, E3 +509470.001}
SPL {X  -162.820, Y  +498.027, Z    +0.000, E1   +21.516, E3 +509482.908}
SPL {X  -162.820, Y  +495.897, Z    +0.000, E1   +21.662, E3 +509492.828}
SPL {X  -162.820, Y  +493.717, Z    +0.000, E1   +21.704, E3 +509503.935}
SPL {X  -162.820, Y  +491.396, Z    +0.000, E1   +21.707, E3 +509516.059}
SPL {X  -162.820, Y  +488.560, Z    +0.000, E1   +21.695, E3 +509531.168}
SPL {X  -162.820, Y  +485.661, Z    +0.000, E1   +21.712, E3 +509546.053}
SPL {X  -162.820, Y  +483.668, Z    +0.000, E1   +21.664, E3 +509556.881}
SPL {X  -162.820, Y  +481.739, Z    +0.000, E1   +21.704, E3 +509566.595}
SPL {X  -162.820, Y  +479.894, Z    +0.000, E1   +21.695, E3 +509576.382}
SPL {X  -162.820, Y  +477.685, Z    +0.000, E1   +21.656, E3 +509588.320}
SPL {X  -162.820, Y  +475.419, Z    +0.000, E1   +21.711, E3 +509599.672}
SPL {X  -162.820, Y  +473.301, Z    +0.000, E1   +21.712, E3 +509610.769}
SPL {X  -162.820, Y  +470.965, Z    +0.000, E1   +21.700, E3 +509623.114}
SPL {X  -162.820, Y  +469.036, Z    +0.000, E1   +21.695, E3 +509633.158}
SPL {X  -162.820, Y  +467.138, Z    +0.000, E1   +21.678, E3 +509643.330}
SPL {X  -162.820, Y  +465.011, Z    +0.000, E1   +21.692, E3 +509654.312}
SPL {X  -162.820, Y  +462.669, Z    +0.000, E1   +21.752, E3 +509666.093}
SPL {X  -162.820, Y  +460.725, Z    +0.000, E1   +21.689, E3 +509676.706}
SPL {X  -162.820, Y  +458.666, Z    +0.000, E1   +21.695, E3 +509687.518}
SPL {X  -162.820, Y  +456.431, Z    +0.000, E1   +21.708, E3 +509699.046}
SPL {X  -162.820, Y  +453.609, Z    +0.000, E1   +21.757, E3 +509713.580}
SPL {X  -162.820, Y  +450.610, Z    +0.000, E1   +21.698, E3 +509729.637}
SPL {X  -162.820, Y  +448.170, Z    +0.000, E1   +21.667, E3 +509742.658}
SPL {X  -162.820, Y  +446.246, Z    +0.000, E1   +21.696, E3 +509752.476}
SPL {X  -162.820, Y  +443.784, Z    +0.000, E1   +21.713, E3 +509765.262}
SPL {X  -162.820, Y  +441.754, Z    +0.000, E1   +21.708, E3 +509775.814}
SPL {X  -162.820, Y  +439.933, Z    +0.000, E1   +21.690, E3 +509785.578}
SPL {X  -162.820, Y  +437.628, Z    +0.000, E1   +21.678, E3 +509797.766}
SPL {X  -162.820, Y  +435.262, Z    +0.000, E1   +21.727, E3 +509809.702}
SPL {X  -162.820, Y  +433.510, Z    +0.000, E1   +21.692, E3 +509819.115}
SPL {X  -162.820, Y  +431.492, Z    +0.000, E1   +21.686, E3 +509829.811}
SPL {X  -162.820, Y  +429.074, Z    +0.000, E1   +21.710, E3 +509842.263}
SPL {X  -162.820, Y  +427.020, Z    +0.000, E1   +21.674, E3 +509853.264}
SPL {X  -162.820, Y  +424.525, Z    +0.000, E1   +21.712, E3 +509866.177}
SPL {X  -162.820, Y  +421.144, Z    +0.000, E1   +21.719, E3 +509883.844}
SPL {X  -162.820, Y  +418.116, Z    +0.000, E1   +21.761, E3 +509899.175}
SPL {X  -162.820, Y  +416.127, Z    +0.000, E1   +21.715, E3 +509909.881}
SPL {X  -162.820, Y  +414.361, Z    +0.000, E1   +21.613, E3 +509920.068}
SPL {X  -162.820, Y  +412.134, Z    +0.000, E1   +21.697, E3 +509931.012}
SPL {X  -162.820, Y  +409.248, Z    +0.000, E1   +21.741, E3 +509945.948}
SPL {X  -162.820, Y  +406.238, Z    +0.000, E1   +21.697, E3 +509961.916}
SPL {X  -162.820, Y  +403.166, Z    +0.000, E1   +21.746, E3 +509977.722}
SPL {X  -162.820, Y  +400.348, Z    +0.000, E1   +21.713, E3 +509992.556}
SPL {X  -162.820, Y  +398.298, Z    +0.000, E1   +21.721, E3 +510003.172}
SPL {X  -162.820, Y  +396.371, Z    +0.000, E1   +21.713, E3 +510013.354}
SPL {X  -162.820, Y  +394.508, Z    +0.000, E1   +21.616, E3 +510023.909}
SPL {X  -162.820, Y  +391.777, Z    +0.000, E1   +21.714, E3 +510037.569}
SPL {X  -162.820, Y  +388.822, Z    +0.000, E1   +21.717, E3 +510052.888}
SPL {X  -162.820, Y  +386.818, Z    +0.000, E1   +21.679, E3 +510063.628}
SPL {X  -162.820, Y  +384.697, Z    +0.000, E1   +21.693, E3 +510074.699}
SPL {X  -162.820, Y  +382.288, Z    +0.000, E1   +21.742, E3 +510086.822}
SPL {X  -162.817, Y  +379.520, Z    +0.000, E1   +21.723, E3 +510101.660}
SPL {X  -162.776, Y  +376.710, Z    +0.000, E1   +21.698, E3 +510116.399}
SPL {X  -162.707, Y  +374.438, Z    +0.000, E1   +21.688, E3 +510128.403}
SPL {X  -162.607, Y  +372.171, Z    +0.000, E1   +21.692, E3 +510140.202}
SPL {X  -162.494, Y  +370.197, Z    +0.000, E1   +21.655, E3 +510150.829}
SPL {X  -162.349, Y  +368.131, Z    +0.000, E1   +21.624, E3 +510161.946}
SPL {X  -162.161, Y  +365.866, Z    +0.000, E1   +21.642, E3 +510173.632}
SPL {X  -161.651, Y  +361.024, Z    +0.000, E1   +22.970, E3 +510187.055}
SPL {X  -160.281, Y  +351.857, Z    +0.000, E1   +24.243, E3 +510222.394}
ENDSPLINE

SPLINE
SPL {X  -161.833, Y  +362.603, Z    +0.000, E1   +17.021, E3 +510237.090}
ENDSPLINE

SPLINE
SPL {X  -160.786, Y  +354.842, Z    +0.000, E1   +19.274, E3 +510269.245}
ENDSPLINE

SPLINE
SPL {X  -162.485, Y  +370.062, Z    +0.000, E1   +10.606, E3 +510275.624}
SPL {X  -162.820, Y  +381.311, Z    +0.000, E1    +4.054, E3 +510265.979}
SPL {X  -162.820, Y  +389.994, Z    +0.000, E1    -2.149, E3 +510260.391}
SPL {X  -162.820, Y  +391.982, Z    +0.000, E1    -3.443, E3 +510270.836}
SPL {X  -162.820, Y  +399.630, Z    +0.000, E1    -9.426, E3 +510273.344}
SPL {X  -162.820, Y  +408.127, Z    +0.000, E1   -18.417, E3 +510259.632}
SPL {X  -162.820, Y  +420.083, Z    +0.000, E1   -24.325, E3 +510280.108}
SPL {X  -162.820, Y  +428.527, Z    +0.000, E1   -26.988, E3 +510297.400}
SPL {X  -162.820, Y  +431.191, Z    +0.000, E1   -23.548, E3 +510332.253}
SPL {X  -162.820, Y  +432.946, Z    +0.000, E1   -22.795, E3 +510346.656}
SPL {X  -162.820, Y  +434.888, Z    +0.000, E1   -22.823, E3 +510356.063}
SPL {X  -162.820, Y  +436.834, Z    +0.000, E1   -22.779, E3 +510366.023}
SPL {X  -162.820, Y  +438.868, Z    +0.000, E1   -22.837, E3 +510375.677}
SPL {X  -162.820, Y  +441.351, Z    +0.000, E1   -22.805, E3 +510388.252}
SPL {X  -162.820, Y  +443.809, Z    +0.000, E1   -22.804, E3 +510400.418}
SPL {X  -162.820, Y  +447.077, Z    +0.000, E1   -22.869, E3 +510416.229}
SPL {X  -162.820, Y  +449.911, Z    +0.000, E1   -22.774, E3 +510430.838}
SPL {X  -162.820, Y  +451.861, Z    +0.000, E1   -22.750, E3 +510440.686}
SPL {X  -162.820, Y  +454.167, Z    +0.000, E1   -22.842, E3 +510451.415}
SPL {X  -162.820, Y  +456.529, Z    +0.000, E1   -22.855, E3 +510462.944}
SPL {X  -162.820, Y  +458.725, Z    +0.000, E1   -22.793, E3 +510474.348}
SPL {X  -162.820, Y  +460.754, Z    +0.000, E1   -22.806, E3 +510484.221}
SPL {X  -162.820, Y  +462.409, Z    +0.000, E1   -22.783, E3 +510492.638}
SPL {X  -162.820, Y  +464.633, Z    +0.000, E1   -22.813, E3 +510503.467}
SPL {X  -162.820, Y  +467.913, Z    +0.000, E1   -22.879, E3 +510519.306}
SPL {X  -162.820, Y  +470.892, Z    +0.000, E1   -22.837, E3 +510534.196}
SPL {X  -162.820, Y  +472.726, Z    +0.000, E1   -22.777, E3 +510543.734}
SPL {X  -162.820, Y  +475.118, Z    +0.000, E1   -22.777, E3 +510555.706}
SPL {X  -162.820, Y  +477.389, Z    +0.000, E1   -22.803, E3 +510566.622}
SPL {X  -162.820, Y  +478.914, Z    +0.000, E1   -22.821, E3 +510574.014}
SPL {X  -162.820, Y  +481.034, Z    +0.000, E1   -22.831, E3 +510584.536}
SPL {X  -162.820, Y  +484.256, Z    +0.000, E1   -22.840, E3 +510600.555}
SPL {X  -162.820, Y  +487.952, Z    +0.000, E1   -22.824, E3 +510618.985}
SPL {X  -162.820, Y  +490.653, Z    +0.000, E1   -22.810, E3 +510632.255}
SPL {X  -162.820, Y  +493.233, Z    +0.000, E1   -22.844, E3 +510644.933}
SPL {X  -162.820, Y  +496.150, Z    +0.000, E1   -22.796, E3 +510659.653}
SPL {X  -162.820, Y  +498.661, Z    +0.000, E1   -22.828, E3 +510671.833}
SPL {X  -162.820, Y  +501.761, Z    +0.000, E1   -22.820, E3 +510687.402}
SPL {X  -162.820, Y  +505.323, Z    +0.000, E1   -22.838, E3 +510704.849}
SPL {X  -162.820, Y  +507.875, Z    +0.000, E1   -22.849, E3 +510717.216}
SPL {X  -162.820, Y  +510.068, Z    +0.000, E1   -22.761, E3 +510728.909}
SPL {X  -162.820, Y  +512.359, Z    +0.000, E1   -22.823, E3 +510739.641}
SPL {X  -162.820, Y  +514.562, Z    +0.000, E1   -22.806, E3 +510750.828}
SPL {X  -162.820, Y  +517.952, Z    +0.000, E1   -22.864, E3 +510767.225}
SPL {X  -162.820, Y  +520.641, Z    +0.000, E1   -22.790, E3 +510780.943}
SPL {X  -162.820, Y  +522.740, Z    +0.000, E1   -22.811, E3 +510791.186}
SPL {X  -162.820, Y  +524.628, Z    +0.000, E1   -22.846, E3 +510800.181}
SPL {X  -162.820, Y  +526.661, Z    +0.000, E1   -22.801, E3 +510810.736}
SPL {X  -162.820, Y  +529.662, Z    +0.000, E1   -22.810, E3 +510825.587}
SPL {X  -162.820, Y  +532.614, Z    +0.000, E1   -22.828, E3 +510839.993}
SPL {X  -162.820, Y  +534.838, Z    +0.000, E1   -22.864, E3 +510850.622}
SPL {X  -162.820, Y  +536.882, Z    +0.000, E1   -22.782, E3 +510861.477}
SPL {X  -162.820, Y  +539.194, Z    +0.000, E1   -22.826, E3 +510872.526}
SPL {X  -162.820, Y  +541.555, Z    +0.000, E1   -22.817, E3 +510884.340}
SPL {X  -162.820, Y  +543.728, Z    +0.000, E1   -22.799, E3 +510895.197}
SPL {X  -162.820, Y  +545.925, Z    +0.000, E1   -22.803, E3 +510906.067}
SPL {X  -162.820, Y  +548.328, Z    +0.000, E1   -22.796, E3 +510918.063}
SPL {X  -162.820, Y  +551.027, Z    +0.000, E1   -22.819, E3 +510931.256}
SPL {X  -162.820, Y  +553.721, Z    +0.000, E1   -22.807, E3 +510944.700}
SPL {X  -162.820, Y  +556.430, Z    +0.000, E1   -22.821, E3 +510957.996}
SPL {X  -162.820, Y  +559.675, Z    +0.000, E1   -22.837, E3 +510974.076}
SPL {X  -162.820, Y  +562.799, Z    +0.000, E1   -22.814, E3 +510989.582}
SPL {X  -162.820, Y  +565.170, Z    +0.000, E1   -22.801, E3 +511001.407}
SPL {X  -162.820, Y  +568.020, Z    +0.000, E1   -22.787, E3 +511015.794}
SPL {X  -162.820, Y  +570.992, Z    +0.000, E1   -22.834, E3 +511030.013}
SPL {X  -162.820, Y  +572.901, Z    +0.000, E1   -22.775, E3 +511039.882}
SPL {X  -162.820, Y  +575.638, Z    +0.000, E1   -22.855, E3 +511052.991}
SPL {X  -162.820, Y  +578.553, Z    +0.000, E1   -22.801, E3 +511067.703}
SPL {X  -162.820, Y  +581.064, Z    +0.000, E1   -22.823, E3 +511079.988}
SPL {X  -162.820, Y  +583.435, Z    +0.000, E1   -22.808, E3 +511091.809}
SPL {X  -162.820, Y  +585.410, Z    +0.000, E1   -22.764, E3 +511101.945}
SPL {X  -162.820, Y  +587.676, Z    +0.000, E1   -22.853, E3 +511112.460}
SPL {X  -162.820, Y  +589.682, Z    +0.000, E1   -22.776, E3 +511122.990}
SPL {X  -162.820, Y  +591.720, Z    +0.000, E1   -22.868, E3 +511132.300}
SPL {X  -162.820, Y  +593.650, Z    +0.000, E1   -22.810, E3 +511142.370}
SPL {X  -162.820, Y  +595.830, Z    +0.000, E1   -22.828, E3 +511152.986}
SPL {X  -162.820, Y  +598.094, Z    +0.000, E1   -22.843, E3 +511164.099}
SPL {X  -162.820, Y  +600.420, Z    +0.000, E1   -22.826, E3 +511175.730}
SPL {X  -162.820, Y  +602.573, Z    +0.000, E1   -22.830, E3 +511186.316}
SPL {X  -162.820, Y  +604.828, Z    +0.000, E1   -22.784, E3 +511197.954}
SPL {X  -162.820, Y  +607.142, Z    +0.000, E1   -22.808, E3 +511209.135}
SPL {X  -162.820, Y  +608.890, Z    +0.000, E1   -22.790, E3 +511217.959}
SPL {X  -162.820, Y  +611.103, Z    +0.000, E1   -22.785, E3 +511228.998}
SPL {X  -162.820, Y  +613.294, Z    +0.000, E1   -22.780, E3 +511239.871}
SPL {X  -162.820, Y  +615.356, Z    +0.000, E1   -22.799, E3 +511249.928}
SPL {X  -162.820, Y  +617.439, Z    +0.000, E1   -22.808, E3 +511260.186}
SPL {X  -162.820, Y  +619.665, Z    +0.000, E1   -22.817, E3 +511271.154}
SPL {X  -162.820, Y  +621.733, Z    +0.000, E1   -22.759, E3 +511281.878}
SPL {X  -162.820, Y  +624.076, Z    +0.000, E1   -22.774, E3 +511293.383}
SPL {X  -162.820, Y  +626.527, Z    +0.000, E1   -22.768, E3 +511305.626}
SPL {X  -162.820, Y  +629.758, Z    +0.000, E1   -22.800, E3 +511321.555}
SPL {X  -162.820, Y  +632.572, Z    +0.000, E1   -22.785, E3 +511335.404}
SPL {X  -162.820, Y  +634.507, Z    +0.000, E1   -22.784, E3 +511345.043}
SPL {X  -162.820, Y  +636.863, Z    +0.000, E1   -22.760, E3 +511356.965}
SPL {X  -162.820, Y  +639.254, Z    +0.000, E1   -22.767, E3 +511368.748}
SPL {X  -162.820, Y  +641.195, Z    +0.000, E1   -22.782, E3 +511378.196}
SPL {X  -162.820, Y  +643.449, Z    +0.000, E1   -22.796, E3 +511389.366}
SPL {X  -162.820, Y  +645.630, Z    +0.000, E1   -22.795, E3 +511400.062}
SPL {X  -162.820, Y  +647.561, Z    +0.000, E1   -22.705, E3 +511410.512}
SPL {X  -162.820, Y  +651.051, Z    +0.000, E1   -22.833, E3 +511426.932}
SPL {X  -162.820, Y  +653.898, Z    +0.000, E1   -22.796, E3 +511441.118}
SPL {X  -162.820, Y  +656.161, Z    +0.000, E1   -22.812, E3 +511452.239}
SPL {X  -162.820, Y  +658.384, Z    +0.000, E1   -22.822, E3 +511463.105}
SPL {X  -162.820, Y  +660.215, Z    +0.000, E1   -22.649, E3 +511473.696}
SPL {X  -162.820, Y  +662.823, Z    +0.000, E1   -22.799, E3 +511485.404}
SPL {X  -162.820, Y  +665.112, Z    +0.000, E1   -22.835, E3 +511496.458}
SPL {X  -162.820, Y  +667.016, Z    +0.000, E1   -22.823, E3 +511505.887}
SPL {X  -162.820, Y  +668.960, Z    +0.000, E1   -22.773, E3 +511516.054}
SPL {X  -162.820, Y  +672.333, Z    +0.000, E1   -22.837, E3 +511532.390}
SPL {X  -162.812, Y  +675.071, Z    +0.000, E1   -22.742, E3 +511546.535}
SPL {X  -162.773, Y  +677.428, Z    +0.000, E1   -22.762, E3 +511558.133}
SPL {X  -162.691, Y  +679.987, Z    +0.000, E1   -22.794, E3 +511570.546}
SPL {X  -162.604, Y  +681.880, Z    +0.000, E1   -22.691, E3 +511580.707}
SPL {X  -162.458, Y  +684.346, Z    +0.000, E1   -22.764, E3 +511592.501}
SPL {X  -162.296, Y  +686.547, Z    +0.000, E1   -22.660, E3 +511604.118}
SPL {X  -162.090, Y  +688.902, Z    +0.000, E1   -22.700, E3 +511615.626}
SPL {X  -161.474, Y  +694.390, Z    +0.000, E1   -24.298, E3 +511628.981}
SPL {X  -158.553, Y  +710.529, Z    +0.000, E1   -30.890, E3 +511645.543}
ENDSPLINE

SPLINE
SPL {X  -161.215, Y  +696.305, Z    +0.000, E1   -20.575, E3 +511672.123}
SPL {X  -161.691, Y  +692.643, Z    +0.000, E1   -17.369, E3 +511688.312}
SPL {X  -162.534, Y  +683.153, Z    +0.000, E1   -10.475, E3 +511713.779}
SPL {X  -162.820, Y  +667.630, Z    +0.000, E1    -0.882, E3 +511707.755}
SPL {X  -162.820, Y  +661.883, Z    +0.000, E1    +3.373, E3 +511713.198}
SPL {X  -162.820, Y  +653.808, Z    +0.000, E1    +9.891, E3 +511710.889}
SPL {X  -162.820, Y  +632.548, Z    +0.000, E1   +27.446, E3 +511707.426}
ENDSPLINE

SPLINE
SPL {X  -162.820, Y  +638.080, Z    +0.000, E1   +18.858, E3 +511735.175}
ENDSPLINE

SPLINE
SPL {X  -162.820, Y  +623.278, Z    +0.000, E1   +28.723, E3 +511736.745}
SPL {X  -162.820, Y  +618.658, Z    +0.000, E1   +26.841, E3 +511765.354}
ENDSPLINE

SPLINE
SPL {X  -162.820, Y  +623.685, Z    +0.000, E1   +22.346, E3 +511777.661}
ENDSPLINE

SPLINE
SPL {X  -162.820, Y  +621.304, Z    +0.000, E1   +22.259, E3 +511790.476}
SPL {X  -162.820, Y  +618.758, Z    +0.000, E1   +22.239, E3 +511803.627}
SPL {X  -162.820, Y  +616.062, Z    +0.000, E1   +22.275, E3 +511817.047}
SPL {X  -162.820, Y  +613.536, Z    +0.000, E1   +22.242, E3 +511830.169}
SPL {X  -162.820, Y  +610.461, Z    +0.000, E1   +22.264, E3 +511845.800}
SPL {X  -162.820, Y  +606.755, Z    +0.000, E1   +22.275, E3 +511864.598}
SPL {X  -162.820, Y  +603.020, Z    +0.000, E1   +22.272, E3 +511883.658}
SPL {X  -162.820, Y  +599.168, Z    +0.000, E1   +22.310, E3 +511902.926}
SPL {X  -162.820, Y  +596.569, Z    +0.000, E1   +22.222, E3 +511916.648}
SPL {X  -162.820, Y  +594.115, Z    +0.000, E1   +22.273, E3 +511928.874}
SPL {X  -162.820, Y  +591.721, Z    +0.000, E1   +22.239, E3 +511941.189}
SPL {X  -162.820, Y  +589.492, Z    +0.000, E1   +22.304, E3 +511952.050}
SPL {X  -162.820, Y  +587.447, Z    +0.000, E1   +22.279, E3 +511962.579}
SPL {X  -162.820, Y  +585.192, Z    +0.000, E1   +22.298, E3 +511973.989}
SPL {X  -162.820, Y  +582.610, Z    +0.000, E1   +22.234, E3 +511987.612}
SPL {X  -162.820, Y  +580.317, Z    +0.000, E1   +22.300, E3 +511998.666}
SPL {X  -162.820, Y  +578.878, Z    +0.000, E1   +22.272, E3 +512006.176}
SPL {X  -162.820, Y  +576.856, Z    +0.000, E1   +22.233, E3 +512016.934}
SPL {X  -162.820, Y  +573.830, Z    +0.000, E1   +22.272, E3 +512032.070}
SPL {X  -162.820, Y  +570.852, Z    +0.000, E1   +22.234, E3 +512047.529}
SPL {X  -162.820, Y  +568.608, Z    +0.000, E1   +22.253, E3 +512058.663}
SPL {X  -162.820, Y  +565.838, Z    +0.000, E1   +22.271, E3 +512072.894}
SPL {X  -162.820, Y  +562.162, Z    +0.000, E1   +22.252, E3 +512091.711}
SPL {X  -162.820, Y  +558.919, Z    +0.000, E1   +22.286, E3 +512107.874}
SPL {X  -162.820, Y  +555.548, Z    +0.000, E1   +22.322, E3 +512124.783}
SPL {X  -162.820, Y  +552.787, Z    +0.000, E1   +22.213, E3 +512139.581}
SPL {X  -162.820, Y  +550.871, Z    +0.000, E1   +22.229, E3 +512149.175}
SPL {X  -162.820, Y  +548.168, Z    +0.000, E1   +22.298, E3 +512162.512}
SPL {X  -162.820, Y  +545.860, Z    +0.000, E1   +22.216, E3 +512174.769}
SPL {X  -162.820, Y  +543.558, Z    +0.000, E1   +22.285, E3 +512186.000}
SPL {X  -162.820, Y  +540.968, Z    +0.000, E1   +22.274, E3 +512199.272}
SPL {X  -162.820, Y  +538.512, Z    +0.000, E1   +22.287, E3 +512211.584}
SPL {X  -162.820, Y  +535.523, Z    +0.000, E1   +22.266, E3 +512227.200}
SPL {X  -162.820, Y  +531.757, Z    +0.000, E1   +22.276, E3 +512246.255}
SPL {X  -162.820, Y  +527.980, Z    +0.000, E1   +22.326, E3 +512265.086}
SPL {X  -162.820, Y  +524.599, Z    +0.000, E1   +22.287, E3 +512282.483}
SPL {X  -162.820, Y  +522.011, Z    +0.000, E1   +22.282, E3 +512295.560}
SPL {X  -162.820, Y  +519.457, Z    +0.000, E1   +22.481, E3 +512306.849}
SPL {X  -162.820, Y  +505.859, Z    +0.000, E1   +28.367, E3 +512321.332}
SPL {X  -162.820, Y  +504.131, Z    +0.000, E1   +27.325, E3 +512335.471}
SPL {X  -162.820, Y  +502.813, Z    +0.000, E1   +26.013, E3 +512350.847}
SPL {X  -162.820, Y  +502.016, Z    +0.000, E1   +24.802, E3 +512363.190}
SPL {X  -162.820, Y  +501.060, Z    +0.000, E1   +24.081, E3 +512373.379}
SPL {X  -162.820, Y  +499.934, Z    +0.000, E1   +22.814, E3 +512389.248}
SPL {X  -162.820, Y  +498.303, Z    +0.000, E1   +21.749, E3 +512406.504}
SPL {X  -162.820, Y  +495.897, Z    +0.000, E1   +21.662, E3 +512419.658}
SPL {X  -162.820, Y  +493.717, Z    +0.000, E1   +21.704, E3 +512430.764}
SPL {X  -162.820, Y  +491.396, Z    +0.000, E1   +21.707, E3 +512442.888}
SPL {X  -162.820, Y  +489.485, Z    +0.000, E1   +21.661, E3 +512453.236}
SPL {X  -162.820, Y  +487.723, Z    +0.000, E1   +21.665, E3 +512462.439}
SPL {X  -162.820, Y  +485.661, Z    +0.000, E1   +21.712, E3 +512472.883}
SPL {X  -162.820, Y  +482.775, Z    +0.000, E1   +21.716, E3 +512488.135}
SPL {X  -162.820, Y  +479.894, Z    +0.000, E1   +21.695, E3 +512503.211}
SPL {X  -162.820, Y  +477.685, Z    +0.000, E1   +21.656, E3 +512515.149}
SPL {X  -162.820, Y  +475.419, Z    +0.000, E1   +21.711, E3 +512526.501}
SPL {X  -162.820, Y  +473.301, Z    +0.000, E1   +21.712, E3 +512537.599}
SPL {X  -162.820, Y  +470.965, Z    +0.000, E1   +21.700, E3 +512549.943}
SPL {X  -162.820, Y  +469.036, Z    +0.000, E1   +21.695, E3 +512559.987}
SPL {X  -162.820, Y  +467.138, Z    +0.000, E1   +21.678, E3 +512570.159}
SPL {X  -162.820, Y  +465.011, Z    +0.000, E1   +21.692, E3 +512581.141}
SPL {X  -162.820, Y  +462.669, Z    +0.000, E1   +21.752, E3 +512592.922}
SPL {X  -162.820, Y  +460.725, Z    +0.000, E1   +21.689, E3 +512603.535}
SPL {X  -162.820, Y  +458.666, Z    +0.000, E1   +21.695, E3 +512614.347}
SPL {X  -162.820, Y  +456.431, Z    +0.000, E1   +21.708, E3 +512625.875}
SPL {X  -162.820, Y  +453.609, Z    +0.000, E1   +21.757, E3 +512640.409}
SPL {X  -162.820, Y  +450.610, Z    +0.000, E1   +21.698, E3 +512656.467}
SPL {X  -162.820, Y  +448.170, Z    +0.000, E1   +21.667, E3 +512669.487}
SPL {X  -162.820, Y  +445.508, Z    +0.000, E1   +21.732, E3 +512683.006}
SPL {X  -162.820, Y  +442.443, Z    +0.000, E1   +21.712, E3 +512699.126}
SPL {X  -162.820, Y  +439.933, Z    +0.000, E1   +21.690, E3 +512712.407}
SPL {X  -162.820, Y  +437.628, Z    +0.000, E1   +21.678, E3 +512724.595}
SPL {X  -162.820, Y  +434.473, Z    +0.000, E1   +21.747, E3 +512740.692}
SPL {X  -162.820, Y  +431.492, Z    +0.000, E1   +21.686, E3 +512756.640}
SPL {X  -162.820, Y  +429.074, Z    +0.000, E1   +21.710, E3 +512769.092}
SPL {X  -162.820, Y  +426.023, Z    +0.000, E1   +21.718, E3 +512785.160}
SPL {X  -162.820, Y  +422.986, Z    +0.000, E1   +21.685, E3 +512801.207}
SPL {X  -162.820, Y  +420.528, Z    +0.000, E1   +21.706, E3 +512813.857}
SPL {X  -162.820, Y  +418.116, Z    +0.000, E1   +21.761, E3 +512826.005}
SPL {X  -162.820, Y  +416.127, Z    +0.000, E1   +21.715, E3 +512836.710}
SPL {X  -162.820, Y  +414.361, Z    +0.000, E1   +21.613, E3 +512846.897}
SPL {X  -162.820, Y  +411.450, Z    +0.000, E1   +21.710, E3 +512861.471}
SPL {X  -162.820, Y  +408.590, Z    +0.000, E1   +21.735, E3 +512876.096}
SPL {X  -162.820, Y  +406.238, Z    +0.000, E1   +21.697, E3 +512888.745}
SPL {X  -162.820, Y  +403.166, Z    +0.000, E1   +21.746, E3 +512904.551}
SPL {X  -162.820, Y  +400.348, Z    +0.000, E1   +21.713, E3 +512919.386}
SPL {X  -162.820, Y  +398.298, Z    +0.000, E1   +21.721, E3 +512930.001}
SPL {X  -162.820, Y  +396.371, Z    +0.000, E1   +21.713, E3 +512940.183}
SPL {X  -162.820, Y  +394.508, Z    +0.000, E1   +21.616, E3 +512950.739}
SPL {X  -162.820, Y  +391.777, Z    +0.000, E1   +21.714, E3 +512964.398}
SPL {X  -162.820, Y  +388.822, Z    +0.000, E1   +21.717, E3 +512979.718}
SPL {X  -162.820, Y  +386.818, Z    +0.000, E1   +21.679, E3 +512990.458}
SPL {X  -162.820, Y  +384.697, Z    +0.000, E1   +21.693, E3 +513001.528}
SPL {X  -162.820, Y  +382.288, Z    +0.000, E1   +21.742, E3 +513013.651}
SPL {X  -162.820, Y  +380.381, Z    +0.000, E1   +21.655, E3 +513024.376}
SPL {X  -162.808, Y  +378.512, Z    +0.000, E1   +21.736, E3 +513033.429}
SPL {X  -162.776, Y  +376.710, Z    +0.000, E1   +21.698, E3 +513043.228}
SPL {X  -162.707, Y  +374.438, Z    +0.000, E1   +21.688, E3 +513055.232}
SPL {X  -162.607, Y  +372.171, Z    +0.000, E1   +21.692, E3 +513067.031}
SPL {X  -162.494, Y  +370.197, Z    +0.000, E1   +21.655, E3 +513077.658}
SPL {X  -162.349, Y  +368.131, Z    +0.000, E1   +21.624, E3 +513088.776}
SPL {X  -162.161, Y  +365.866, Z    +0.000, E1   +21.642, E3 +513100.461}
SPL {X  -161.927, Y  +363.466, Z    +0.000, E1   +21.730, E3 +513112.232}
SPL {X  -160.290, Y  +351.907, Z    +0.000, E1   +27.562, E3 +513119.810}
SPL {X  -159.725, Y  +348.905, Z    +0.000, E1   +26.136, E3 +513145.045}
ENDSPLINE

SPLINE
SPL {X  -160.871, Y  +355.385, Z    +0.000, E1   +21.841, E3 +513153.888}
SPL {X  -161.833, Y  +362.603, Z    +0.000, E1   +17.021, E3 +513163.919}
ENDSPLINE

SPLINE
SPL {X  -160.786, Y  +354.842, Z    +0.000, E1   +19.274, E3 +513196.075}
ENDSPLINE

SPLINE
SPL {X  -162.485, Y  +370.062, Z    +0.000, E1   +10.606, E3 +513202.453}
SPL {X  -162.820, Y  +381.311, Z    +0.000, E1    +4.054, E3 +513192.808}
SPL {X  -162.820, Y  +389.994, Z    +0.000, E1    -2.149, E3 +513187.220}
SPL {X  -162.820, Y  +391.982, Z    +0.000, E1    -3.443, E3 +513197.666}
SPL {X  -162.820, Y  +399.630, Z    +0.000, E1    -9.426, E3 +513200.173}
SPL {X  -162.820, Y  +408.127, Z    +0.000, E1   -18.417, E3 +513186.462}
SPL {X  -162.820, Y  +420.083, Z    +0.000, E1   -24.325, E3 +513206.937}
SPL {X  -162.820, Y  +428.527, Z    +0.000, E1   -26.988, E3 +513224.229}
SPL {X  -162.820, Y  +431.336, Z    +0.000, E1   -24.162, E3 +513254.439}
SPL {X  -162.820, Y  +432.048, Z    +0.000, E1   -22.832, E3 +513268.943}
SPL {X  -162.820, Y  +434.888, Z    +0.000, E1   -22.823, E3 +513282.892}
SPL {X  -162.820, Y  +436.834, Z    +0.000, E1   -22.779, E3 +513292.852}
SPL {X  -162.820, Y  +438.868, Z    +0.000, E1   -22.837, E3 +513302.506}
SPL {X  -162.820, Y  +441.351, Z    +0.000, E1   -22.805, E3 +513315.081}
SPL {X  -162.820, Y  +443.809, Z    +0.000, E1   -22.804, E3 +513327.248}
SPL {X  -162.820, Y  +447.077, Z    +0.000, E1   -22.869, E3 +513343.058}
SPL {X  -162.820, Y  +449.911, Z    +0.000, E1   -22.774, E3 +513357.668}
SPL {X  -162.820, Y  +451.861, Z    +0.000, E1   -22.750, E3 +513367.515}
SPL {X  -162.820, Y  +454.167, Z    +0.000, E1   -22.842, E3 +513378.245}
SPL {X  -162.820, Y  +456.529, Z    +0.000, E1   -22.855, E3 +513389.773}
SPL {X  -162.820, Y  +458.725, Z    +0.000, E1   -22.793, E3 +513401.177}
SPL {X  -162.820, Y  +460.754, Z    +0.000, E1   -22.806, E3 +513411.050}
SPL {X  -162.820, Y  +462.409, Z    +0.000, E1   -22.783, E3 +513419.467}
SPL {X  -162.820, Y  +464.633, Z    +0.000, E1   -22.813, E3 +513430.297}
SPL {X  -162.820, Y  +467.913, Z    +0.000, E1   -22.879, E3 +513446.136}
SPL {X  -162.820, Y  +470.892, Z    +0.000, E1   -22.837, E3 +513461.025}
SPL {X  -162.820, Y  +472.726, Z    +0.000, E1   -22.777, E3 +513470.564}
SPL {X  -162.820, Y  +475.118, Z    +0.000, E1   -22.777, E3 +513482.535}
SPL {X  -162.820, Y  +478.177, Z    +0.000, E1   -22.834, E3 +513497.228}
SPL {X  -162.820, Y  +481.034, Z    +0.000, E1   -22.831, E3 +513511.365}
SPL {X  -162.820, Y  +483.391, Z    +0.000, E1   -22.793, E3 +513523.302}
SPL {X  -162.820, Y  +486.307, Z    +0.000, E1   -22.833, E3 +513537.555}
SPL {X  -162.820, Y  +488.828, Z    +0.000, E1   -22.793, E3 +513550.198}
SPL {X  -162.820, Y  +491.768, Z    +0.000, E1   -22.852, E3 +513564.495}
SPL {X  -162.820, Y  +495.526, Z    +0.000, E1   -22.833, E3 +513583.266}
SPL {X  -162.820, Y  +499.330, Z    +0.000, E1   -22.841, E3 +513602.048}
SPL {X  -162.820, Y  +503.049, Z    +0.000, E1   -22.823, E3 +513620.597}
SPL {X  -162.820, Y  +506.908, Z    +0.000, E1   -22.877, E3 +513639.267}
SPL {X  -162.820, Y  +510.068, Z    +0.000, E1   -22.761, E3 +513655.738}
SPL {X  -162.820, Y  +512.359, Z    +0.000, E1   -22.823, E3 +513666.470}
SPL {X  -162.820, Y  +514.562, Z    +0.000, E1   -22.806, E3 +513677.657}
SPL {X  -162.820, Y  +517.952, Z    +0.000, E1   -22.864, E3 +513694.054}
SPL {X  -162.820, Y  +520.641, Z    +0.000, E1   -22.790, E3 +513707.773}
SPL {X  -162.820, Y  +522.740, Z    +0.000, E1   -22.811, E3 +513718.015}
SPL {X  -162.820, Y  +524.628, Z    +0.000, E1   -22.846, E3 +513727.010}
SPL {X  -162.820, Y  +526.661, Z    +0.000, E1   -22.801, E3 +513737.566}
SPL {X  -162.820, Y  +529.662, Z    +0.000, E1   -22.810, E3 +513752.416}
SPL {X  -162.820, Y  +532.614, Z    +0.000, E1   -22.828, E3 +513766.823}
SPL {X  -162.820, Y  +534.838, Z    +0.000, E1   -22.864, E3 +513777.451}
SPL {X  -162.820, Y  +536.882, Z    +0.000, E1   -22.782, E3 +513788.306}
SPL {X  -162.820, Y  +539.194, Z    +0.000, E1   -22.826, E3 +513799.355}
SPL {X  -162.820, Y  +541.555, Z    +0.000, E1   -22.817, E3 +513811.169}
SPL {X  -162.820, Y  +543.728, Z    +0.000, E1   -22.799, E3 +513822.027}
SPL {X  -162.820, Y  +545.925, Z    +0.000, E1   -22.803, E3 +513832.897}
SPL {X  -162.820, Y  +548.328, Z    +0.000, E1   -22.796, E3 +513844.892}
SPL {X  -162.820, Y  +551.027, Z    +0.000, E1   -22.819, E3 +513858.085}
SPL {X  -162.820, Y  +553.721, Z    +0.000, E1   -22.807, E3 +513871.529}
SPL {X  -162.820, Y  +556.430, Z    +0.000, E1   -22.821, E3 +513884.825}
SPL {X  -162.820, Y  +559.675, Z    +0.000, E1   -22.837, E3 +513900.905}
SPL {X  -162.820, Y  +562.799, Z    +0.000, E1   -22.814, E3 +513916.412}
SPL {X  -162.820, Y  +565.170, Z    +0.000, E1   -22.801, E3 +513928.236}
SPL {X  -162.820, Y  +568.020, Z    +0.000, E1   -22.787, E3 +513942.623}
SPL {X  -162.820, Y  +570.992, Z    +0.000, E1   -22.834, E3 +513956.842}
SPL {X  -162.820, Y  +572.901, Z    +0.000, E1   -22.775, E3 +513966.711}
SPL {X  -162.820, Y  +575.638, Z    +0.000, E1   -22.855, E3 +513979.820}
SPL {X  -162.820, Y  +578.553, Z    +0.000, E1   -22.801, E3 +513994.533}
SPL {X  -162.820, Y  +581.064, Z    +0.000, E1   -22.823, E3 +514006.817}
SPL {X  -162.820, Y  +583.435, Z    +0.000, E1   -22.808, E3 +514018.639}
SPL {X  -162.820, Y  +585.410, Z    +0.000, E1   -22.764, E3 +514028.774}
SPL {X  -162.820, Y  +587.676, Z    +0.000, E1   -22.853, E3 +514039.289}
SPL {X  -162.820, Y  +589.682, Z    +0.000, E1   -22.776, E3 +514049.819}
SPL {X  -162.820, Y  +591.720, Z    +0.000, E1   -22.868, E3 +514059.130}
SPL {X  -162.820, Y  +593.650, Z    +0.000, E1   -22.810, E3 +514069.200}
SPL {X  -162.820, Y  +595.830, Z    +0.000, E1   -22.828, E3 +514079.815}
SPL {X  -162.820, Y  +598.094, Z    +0.000, E1   -22.843, E3 +514090.928}
SPL {X  -162.820, Y  +600.420, Z    +0.000, E1   -22.826, E3 +514102.560}
SPL {X  -162.820, Y  +602.573, Z    +0.000, E1   -22.830, E3 +514113.145}
SPL {X  -162.820, Y  +604.828, Z    +0.000, E1   -22.784, E3 +514124.783}
SPL {X  -162.820, Y  +608.133, Z    +0.000, E1   -22.831, E3 +514140.901}
SPL {X  -162.820, Y  +611.103, Z    +0.000, E1   -22.785, E3 +514155.827}
SPL {X  -162.820, Y  +613.294, Z    +0.000, E1   -22.780, E3 +514166.700}
SPL {X  -162.820, Y  +615.356, Z    +0.000, E1   -22.799, E3 +514176.757}
SPL {X  -162.820, Y  +617.439, Z    +0.000, E1   -22.808, E3 +514187.015}
SPL {X  -162.820, Y  +619.665, Z    +0.000, E1   -22.817, E3 +514197.983}
SPL {X  -162.820, Y  +621.733, Z    +0.000, E1   -22.759, E3 +514208.707}
SPL {X  -162.820, Y  +624.076, Z    +0.000, E1   -22.774, E3 +514220.213}
SPL {X  -162.820, Y  +626.527, Z    +0.000, E1   -22.768, E3 +514232.455}
SPL {X  -162.820, Y  +629.758, Z    +0.000, E1   -22.800, E3 +514248.384}
SPL {X  -162.820, Y  +632.572, Z    +0.000, E1   -22.785, E3 +514262.233}
SPL {X  -162.820, Y  +634.507, Z    +0.000, E1   -22.784, E3 +514271.872}
SPL {X  -162.820, Y  +636.863, Z    +0.000, E1   -22.760, E3 +514283.794}
SPL {X  -162.820, Y  +640.111, Z    +0.000, E1   -22.809, E3 +514299.677}
SPL {X  -162.820, Y  +643.449, Z    +0.000, E1   -22.796, E3 +514316.195}
SPL {X  -162.820, Y  +645.630, Z    +0.000, E1   -22.795, E3 +514326.891}
SPL {X  -162.820, Y  +647.561, Z    +0.000, E1   -22.705, E3 +514337.342}
SPL {X  -162.820, Y  +649.758, Z    +0.000, E1   -22.780, E3 +514347.532}
SPL {X  -162.820, Y  +651.708, Z    +0.000, E1   -22.810, E3 +514357.026}
SPL {X  -162.820, Y  +653.898, Z    +0.000, E1   -22.796, E3 +514367.947}
SPL {X  -162.820, Y  +656.161, Z    +0.000, E1   -22.812, E3 +514379.068}
SPL {X  -162.820, Y  +658.384, Z    +0.000, E1   -22.822, E3 +514389.935}
SPL {X  -162.820, Y  +660.215, Z    +0.000, E1   -22.649, E3 +514400.525}
SPL {X  -162.820, Y  +662.823, Z    +0.000, E1   -22.799, E3 +514412.233}
SPL {X  -162.820, Y  +665.112, Z    +0.000, E1   -22.835, E3 +514423.288}
SPL {X  -162.820, Y  +667.016, Z    +0.000, E1   -22.823, E3 +514432.716}
SPL {X  -162.820, Y  +668.960, Z    +0.000, E1   -22.773, E3 +514442.884}
SPL {X  -162.820, Y  +672.333, Z    +0.000, E1   -22.837, E3 +514459.220}
SPL {X  -162.812, Y  +675.071, Z    +0.000, E1   -22.742, E3 +514473.365}
SPL {X  -162.773, Y  +677.428, Z    +0.000, E1   -22.762, E3 +514484.962}
SPL {X  -162.691, Y  +679.987, Z    +0.000, E1   -22.794, E3 +514497.375}
SPL {X  -162.604, Y  +681.880, Z    +0.000, E1   -22.691, E3 +514507.536}
SPL {X  -162.458, Y  +684.346, Z    +0.000, E1   -22.764, E3 +514519.330}
SPL {X  -162.296, Y  +686.547, Z    +0.000, E1   -22.660, E3 +514530.947}
SPL {X  -162.164, Y  +688.106, Z    +0.000, E1   -22.661, E3 +514538.680}
SPL {X  -161.938, Y  +690.422, Z    +0.000, E1   -22.769, E3 +514549.356}
SPL {X  -161.065, Y  +697.344, Z    +0.000, E1   -25.698, E3 +514558.475}
SPL {X  -158.730, Y  +709.763, Z    +0.000, E1   -31.225, E3 +514567.149}
ENDSPLINE

SPLINE
SPL {X  -160.932, Y  +698.225, Z    +0.000, E1   -21.712, E3 +514598.258}
SPL {X  -161.917, Y  +690.622, Z    +0.000, E1   -16.445, E3 +514611.859}
ENDSPLINE

SPLINE
SPL {X  -161.349, Y  +695.340, Z    +0.000, E1   -18.625, E3 +514619.477}
ENDSPLINE

SPLINE
SPL {X  -162.534, Y  +683.153, Z    +0.000, E1   -10.475, E3 +514640.608}
SPL {X  -162.820, Y  +667.630, Z    +0.000, E1    -0.882, E3 +514634.584}
SPL {X  -162.820, Y  +661.883, Z    +0.000, E1    +3.373, E3 +514640.027}
SPL {X  -162.820, Y  +655.163, Z    +0.000, E1    +8.702, E3 +514639.626}
SPL {X  -162.820, Y  +634.515, Z    +0.000, E1   +26.439, E3 +514632.039}
ENDSPLINE

SPLINE
SPL {X  -162.820, Y  +638.080, Z    +0.000, E1   +18.858, E3 +514662.004}
ENDSPLINE

SPLINE
SPL {X  -162.820, Y  +623.278, Z    +0.000, E1   +28.723, E3 +514663.574}
SPL {X  -162.820, Y  +618.658, Z    +0.000, E1   +26.841, E3 +514692.183}
ENDSPLINE

SPLINE
SPL {X  -162.820, Y  +623.685, Z    +0.000, E1   +22.346, E3 +514704.490}
ENDSPLINE

SPLINE
SPL {X  -162.820, Y  +621.304, Z    +0.000, E1   +22.259, E3 +514717.305}
SPL {X  -162.820, Y  +618.758, Z    +0.000, E1   +22.239, E3 +514730.456}
SPL {X  -162.820, Y  +616.062, Z    +0.000, E1   +22.275, E3 +514743.877}
SPL {X  -162.820, Y  +613.536, Z    +0.000, E1   +22.242, E3 +514756.998}
SPL {X  -162.820, Y  +611.128, Z    +0.000, E1   +22.252, E3 +514769.169}
SPL {X  -162.820, Y  +608.428, Z    +0.000, E1   +22.255, E3 +514782.952}
SPL {X  -162.820, Y  +605.984, Z    +0.000, E1   +22.221, E3 +514795.589}
SPL {X  -162.820, Y  +603.020, Z    +0.000, E1   +22.272, E3 +514810.487}
SPL {X  -162.820, Y  +599.168, Z    +0.000, E1   +22.310, E3 +514829.755}
SPL {X  -162.820, Y  +595.597, Z    +0.000, E1   +22.284, E3 +514848.091}
SPL {X  -162.820, Y  +592.389, Z    +0.000, E1   +22.245, E3 +514864.695}
SPL {X  -162.820, Y  +589.492, Z    +0.000, E1   +22.304, E3 +514878.879}
SPL {X  -162.820, Y  +587.447, Z    +0.000, E1   +22.279, E3 +514889.408}
SPL {X  -162.820, Y  +585.192, Z    +0.000, E1   +22.298, E3 +514900.818}
SPL {X  -162.820, Y  +582.610, Z    +0.000, E1   +22.234, E3 +514914.442}
SPL {X  -162.820, Y  +579.691, Z    +0.000, E1   +22.312, E3 +514928.713}
SPL {X  -162.820, Y  +577.460, Z    +0.000, E1   +22.218, E3 +514940.700}
SPL {X  -162.820, Y  +575.394, Z    +0.000, E1   +22.240, E3 +514951.125}
SPL {X  -162.820, Y  +572.645, Z    +0.000, E1   +22.246, E3 +514965.122}
SPL {X  -162.820, Y  +570.282, Z    +0.000, E1   +22.231, E3 +514977.173}
SPL {X  -162.820, Y  +567.961, Z    +0.000, E1   +22.247, E3 +514988.962}
SPL {X  -162.820, Y  +564.506, Z    +0.000, E1   +22.298, E3 +515006.277}
SPL {X  -162.820, Y  +561.620, Z    +0.000, E1   +22.191, E3 +515021.658}
SPL {X  -162.820, Y  +559.515, Z    +0.000, E1   +22.273, E3 +515031.659}
SPL {X  -162.820, Y  +556.723, Z    +0.000, E1   +22.309, E3 +515045.743}
SPL {X  -162.820, Y  +553.294, Z    +0.000, E1   +22.266, E3 +515063.531}
SPL {X  -162.820, Y  +550.871, Z    +0.000, E1   +22.229, E3 +515076.005}
SPL {X  -162.820, Y  +548.168, Z    +0.000, E1   +22.298, E3 +515089.341}
SPL {X  -162.820, Y  +545.860, Z    +0.000, E1   +22.216, E3 +515101.599}
SPL {X  -162.820, Y  +543.558, Z    +0.000, E1   +22.285, E3 +515112.829}
SPL {X  -162.820, Y  +540.968, Z    +0.000, E1   +22.274, E3 +515126.101}
SPL {X  -162.820, Y  +538.512, Z    +0.000, E1   +22.287, E3 +515138.414}
SPL {X  -162.820, Y  +535.523, Z    +0.000, E1   +22.266, E3 +515154.029}
SPL {X  -162.820, Y  +531.757, Z    +0.000, E1   +22.276, E3 +515173.084}
SPL {X  -162.820, Y  +527.980, Z    +0.000, E1   +22.326, E3 +515191.915}
SPL {X  -162.820, Y  +524.599, Z    +0.000, E1   +22.287, E3 +515209.312}
SPL {X  -162.820, Y  +522.011, Z    +0.000, E1   +22.282, E3 +515222.389}
SPL {X  -162.820, Y  +519.457, Z    +0.000, E1   +22.481, E3 +515233.679}
SPL {X  -162.820, Y  +505.859, Z    +0.000, E1   +28.367, E3 +515248.162}
SPL {X  -162.820, Y  +504.131, Z    +0.000, E1   +27.325, E3 +515262.300}
SPL {X  -162.820, Y  +503.215, Z    +0.000, E1   +26.369, E3 +515272.986}
SPL {X  -162.820, Y  +502.502, Z    +0.000, E1   +25.597, E3 +515281.832}
SPL {X  -162.820, Y  +501.672, Z    +0.000, E1   +24.583, E3 +515293.447}
SPL {X  -162.820, Y  +500.515, Z    +0.000, E1   +23.444, E3 +515307.978}
SPL {X  -162.820, Y  +499.633, Z    +0.000, E1   +22.486, E3 +515320.023}
SPL {X  -162.820, Y  +498.303, Z    +0.000, E1   +21.749, E3 +515333.333}
SPL {X  -162.820, Y  +495.897, Z    +0.000, E1   +21.662, E3 +515346.487}
SPL {X  -162.820, Y  +493.717, Z    +0.000, E1   +21.704, E3 +515357.593}
SPL {X  -162.820, Y  +491.396, Z    +0.000, E1   +21.707, E3 +515369.717}
SPL {X  -162.820, Y  +489.485, Z    +0.000, E1   +21.661, E3 +515380.065}
SPL {X  -162.820, Y  +487.723, Z    +0.000, E1   +21.665, E3 +515389.268}
SPL {X  -162.820, Y  +485.661, Z    +0.000, E1   +21.712, E3 +515399.712}
SPL {X  -162.820, Y  +482.775, Z    +0.000, E1   +21.716, E3 +515414.964}
SPL {X  -162.820, Y  +479.894, Z    +0.000, E1   +21.695, E3 +515430.040}
SPL {X  -162.820, Y  +477.685, Z    +0.000, E1   +21.656, E3 +515441.978}
SPL {X  -162.820, Y  +475.419, Z    +0.000, E1   +21.711, E3 +515453.331}
SPL {X  -162.820, Y  +473.301, Z    +0.000, E1   +21.712, E3 +515464.428}
SPL {X  -162.820, Y  +470.965, Z    +0.000, E1   +21.700, E3 +515476.773}
SPL {X  -162.820, Y  +469.036, Z    +0.000, E1   +21.695, E3 +515486.817}
SPL {X  -162.820, Y  +467.138, Z    +0.000, E1   +21.678, E3 +515496.988}
SPL {X  -162.820, Y  +465.011, Z    +0.000, E1   +21.692, E3 +515507.971}
SPL {X  -162.820, Y  +462.669, Z    +0.000, E1   +21.752, E3 +515519.751}
SPL {X  -162.820, Y  +460.725, Z    +0.000, E1   +21.689, E3 +515530.364}
SPL {X  -162.820, Y  +458.666, Z    +0.000, E1   +21.695, E3 +515541.176}
SPL {X  -162.820, Y  +456.431, Z    +0.000, E1   +21.708, E3 +515552.705}
SPL {X  -162.820, Y  +454.628, Z    +0.000, E1   +21.674, E3 +515562.423}
SPL {X  -162.820, Y  +452.690, Z    +0.000, E1   +21.773, E3 +515571.697}
SPL {X  -162.820, Y  +450.610, Z    +0.000, E1   +21.698, E3 +515583.296}
SPL {X  -162.820, Y  +448.170, Z    +0.000, E1   +21.667, E3 +515596.317}
SPL {X  -162.820, Y  +446.246, Z    +0.000, E1   +21.696, E3 +515606.134}
SPL {X  -162.820, Y  +443.784, Z    +0.000, E1   +21.713, E3 +515618.921}
SPL {X  -162.820, Y  +441.754, Z    +0.000, E1   +21.708, E3 +515629.473}
SPL {X  -162.820, Y  +439.933, Z    +0.000, E1   +21.690, E3 +515639.236}
SPL {X  -162.820, Y  +437.628, Z    +0.000, E1   +21.678, E3 +515651.424}
SPL {X  -162.820, Y  +434.473, Z    +0.000, E1   +21.747, E3 +515667.521}
SPL {X  -162.820, Y  +431.492, Z    +0.000, E1   +21.686, E3 +515683.469}
SPL {X  -162.820, Y  +429.074, Z    +0.000, E1   +21.710, E3 +515695.921}
SPL {X  -162.820, Y  +426.023, Z    +0.000, E1   +21.718, E3 +515711.989}
SPL {X  -162.820, Y  +422.986, Z    +0.000, E1   +21.685, E3 +515728.037}
SPL {X  -162.820, Y  +420.528, Z    +0.000, E1   +21.706, E3 +515740.687}
SPL {X  -162.820, Y  +418.116, Z    +0.000, E1   +21.761, E3 +515752.834}
SPL {X  -162.820, Y  +416.127, Z    +0.000, E1   +21.715, E3 +515763.539}
SPL {X  -162.820, Y  +414.361, Z    +0.000, E1   +21.613, E3 +515773.726}
SPL {X  -162.820, Y  +411.450, Z    +0.000, E1   +21.710, E3 +515788.300}
SPL {X  -162.820, Y  +408.590, Z    +0.000, E1   +21.735, E3 +515802.925}
SPL {X  -162.820, Y  +406.238, Z    +0.000, E1   +21.697, E3 +515815.574}
SPL {X  -162.820, Y  +403.166, Z    +0.000, E1   +21.746, E3 +515831.380}
SPL {X  -162.820, Y  +400.348, Z    +0.000, E1   +21.713, E3 +515846.215}
SPL {X  -162.820, Y  +398.298, Z    +0.000, E1   +21.721, E3 +515856.831}
SPL {X  -162.820, Y  +396.371, Z    +0.000, E1   +21.713, E3 +515867.012}
SPL {X  -162.820, Y  +394.508, Z    +0.000, E1   +21.616, E3 +515877.568}
SPL {X  -162.820, Y  +391.777, Z    +0.000, E1   +21.714, E3 +515891.227}
SPL {X  -162.820, Y  +388.822, Z    +0.000, E1   +21.717, E3 +515906.547}
SPL {X  -162.820, Y  +386.818, Z    +0.000, E1   +21.679, E3 +515917.287}
SPL {X  -162.820, Y  +384.697, Z    +0.000, E1   +21.693, E3 +515928.357}
SPL {X  -162.820, Y  +382.288, Z    +0.000, E1   +21.742, E3 +515940.481}
SPL {X  -162.817, Y  +379.520, Z    +0.000, E1   +21.723, E3 +515955.318}
SPL {X  -162.776, Y  +376.710, Z    +0.000, E1   +21.698, E3 +515970.057}
SPL {X  -162.707, Y  +374.438, Z    +0.000, E1   +21.688, E3 +515982.061}
SPL {X  -162.607, Y  +372.171, Z    +0.000, E1   +21.692, E3 +515993.861}
SPL {X  -162.494, Y  +370.197, Z    +0.000, E1   +21.655, E3 +516004.487}
SPL {X  -162.349, Y  +368.131, Z    +0.000, E1   +21.624, E3 +516015.605}
SPL {X  -162.161, Y  +365.866, Z    +0.000, E1   +21.642, E3 +516027.290}
SPL {X  -161.651, Y  +361.024, Z    +0.000, E1   +22.970, E3 +516040.713}
SPL {X  -160.281, Y  +351.857, Z    +0.000, E1   +24.243, E3 +516076.053}
ENDSPLINE

SPLINE
SPL {X  -161.833, Y  +362.603, Z    +0.000, E1   +17.021, E3 +516090.748}
ENDSPLINE

SPLINE
SPL {X  -160.786, Y  +354.842, Z    +0.000, E1   +19.274, E3 +516122.904}
ENDSPLINE

SPLINE
SPL {X  -162.485, Y  +370.062, Z    +0.000, E1   +10.606, E3 +516129.282}
SPL {X  -162.818, Y  +379.636, Z    +0.000, E1    +5.115, E3 +516118.631}
SPL {X  -162.820, Y  +386.976, Z    +0.000, E1    +0.144, E3 +516117.730}
SPL {X  -162.820, Y  +391.982, Z    +0.000, E1    -3.443, E3 +516124.495}
SPL {X  -162.820, Y  +399.630, Z    +0.000, E1    -9.426, E3 +516127.002}
SPL {X  -162.820, Y  +408.127, Z    +0.000, E1   -18.417, E3 +516113.291}
SPL {X  -162.820, Y  +420.083, Z    +0.000, E1   -24.325, E3 +516133.766}
SPL {X  -162.820, Y  +428.527, Z    +0.000, E1   -26.988, E3 +516151.058}
SPL {X  -162.820, Y  +431.191, Z    +0.000, E1   -23.548, E3 +516185.911}
SPL {X  -162.820, Y  +432.946, Z    +0.000, E1   -22.795, E3 +516200.315}
SPL {X  -162.820, Y  +434.888, Z    +0.000, E1   -22.823, E3 +516209.722}
SPL {X  -162.820, Y  +436.834, Z    +0.000, E1   -22.779, E3 +516219.682}
SPL {X  -162.820, Y  +438.868, Z    +0.000, E1   -22.837, E3 +516229.335}
SPL {X  -162.820, Y  +441.351, Z    +0.000, E1   -22.805, E3 +516241.911}
SPL {X  -162.820, Y  +443.809, Z    +0.000, E1   -22.804, E3 +516254.077}
SPL {X  -162.820, Y  +446.105, Z    +0.000, E1   -22.815, E3 +516265.319}
SPL {X  -162.820, Y  +447.974, Z    +0.000, E1   -22.856, E3 +516274.222}
SPL {X  -162.820, Y  +449.911, Z    +0.000, E1   -22.774, E3 +516284.497}
SPL {X  -162.820, Y  +451.861, Z    +0.000, E1   -22.750, E3 +516294.344}
SPL {X  -162.820, Y  +454.167, Z    +0.000, E1   -22.842, E3 +516305.074}
SPL {X  -162.820, Y  +456.529, Z    +0.000, E1   -22.855, E3 +516316.602}
SPL {X  -162.820, Y  +458.725, Z    +0.000, E1   -22.793, E3 +516328.007}
SPL {X  -162.820, Y  +460.754, Z    +0.000, E1   -22.806, E3 +516337.880}
SPL {X  -162.820, Y  +462.409, Z    +0.000, E1   -22.783, E3 +516346.296}
SPL {X  -162.820, Y  +464.633, Z    +0.000, E1   -22.813, E3 +516357.126}
SPL {X  -162.820, Y  +467.913, Z    +0.000, E1   -22.879, E3 +516372.965}
SPL {X  -162.820, Y  +470.892, Z    +0.000, E1   -22.837, E3 +516387.854}
SPL {X  -162.820, Y  +472.726, Z    +0.000, E1   -22.777, E3 +516397.393}
SPL {X  -162.820, Y  +475.118, Z    +0.000, E1   -22.777, E3 +516409.364}
SPL {X  -162.820, Y  +477.389, Z    +0.000, E1   -22.803, E3 +516420.281}
SPL {X  -162.820, Y  +478.914, Z    +0.000, E1   -22.821, E3 +516427.673}
SPL {X  -162.820, Y  +481.034, Z    +0.000, E1   -22.831, E3 +516438.195}
SPL {X  -162.820, Y  +484.256, Z    +0.000, E1   -22.840, E3 +516454.213}
SPL {X  -162.820, Y  +487.952, Z    +0.000, E1   -22.824, E3 +516472.644}
SPL {X  -162.820, Y  +491.768, Z    +0.000, E1   -22.852, E3 +516491.325}
SPL {X  -162.820, Y  +495.526, Z    +0.000, E1   -22.833, E3 +516510.096}
SPL {X  -162.820, Y  +499.330, Z    +0.000, E1   -22.841, E3 +516528.877}
SPL {X  -162.820, Y  +503.049, Z    +0.000, E1   -22.823, E3 +516547.426}
SPL {X  -162.820, Y  +506.908, Z    +0.000, E1   -22.877, E3 +516566.096}
SPL {X  -162.820, Y  +510.068, Z    +0.000, E1   -22.761, E3 +516582.568}
SPL {X  -162.820, Y  +512.359, Z    +0.000, E1   -22.823, E3 +516593.299}
SPL {X  -162.820, Y  +513.873, Z    +0.000, E1   -22.800, E3 +516600.986}
SPL {X  -162.820, Y  +516.100, Z    +0.000, E1   -22.809, E3 +516612.062}
SPL {X  -162.820, Y  +518.662, Z    +0.000, E1   -22.847, E3 +516624.361}
SPL {X  -162.820, Y  +520.641, Z    +0.000, E1   -22.790, E3 +516634.602}
SPL {X  -162.820, Y  +523.535, Z    +0.000, E1   -22.857, E3 +516648.571}
SPL {X  -162.820, Y  +526.661, Z    +0.000, E1   -22.801, E3 +516664.395}
SPL {X  -162.820, Y  +528.725, Z    +0.000, E1   -22.770, E3 +516674.764}
SPL {X  -162.820, Y  +530.303, Z    +0.000, E1   -22.798, E3 +516682.383}
SPL {X  -162.820, Y  +532.614, Z    +0.000, E1   -22.828, E3 +516693.652}
SPL {X  -162.820, Y  +534.838, Z    +0.000, E1   -22.864, E3 +516704.281}
SPL {X  -162.820, Y  +536.882, Z    +0.000, E1   -22.782, E3 +516715.136}
SPL {X  -162.820, Y  +539.194, Z    +0.000, E1   -22.826, E3 +516726.184}
SPL {X  -162.820, Y  +541.555, Z    +0.000, E1   -22.817, E3 +516737.999}
SPL {X  -162.820, Y  +543.728, Z    +0.000, E1   -22.799, E3 +516748.856}
SPL {X  -162.820, Y  +545.925, Z    +0.000, E1   -22.803, E3 +516759.726}
SPL {X  -162.820, Y  +549.071, Z    +0.000, E1   -22.836, E3 +516775.253}
SPL {X  -162.820, Y  +553.089, Z    +0.000, E1   -22.838, E3 +516795.153}
SPL {X  -162.820, Y  +556.430, Z    +0.000, E1   -22.821, E3 +516811.654}
SPL {X  -162.820, Y  +559.675, Z    +0.000, E1   -22.837, E3 +516827.735}
SPL {X  -162.820, Y  +562.799, Z    +0.000, E1   -22.814, E3 +516843.241}
SPL {X  -162.820, Y  +565.170, Z    +0.000, E1   -22.801, E3 +516855.066}
SPL {X  -162.820, Y  +568.020, Z    +0.000, E1   -22.787, E3 +516869.452}
SPL {X  -162.820, Y  +570.992, Z    +0.000, E1   -22.834, E3 +516883.672}
SPL {X  -162.820, Y  +572.901, Z    +0.000, E1   -22.775, E3 +516893.540}
SPL {X  -162.820, Y  +575.638, Z    +0.000, E1   -22.855, E3 +516906.649}
SPL {X  -162.820, Y  +578.553, Z    +0.000, E1   -22.801, E3 +516921.362}
SPL {X  -162.820, Y  +581.064, Z    +0.000, E1   -22.823, E3 +516933.646}
SPL {X  -162.820, Y  +583.435, Z    +0.000, E1   -22.808, E3 +516945.468}
SPL {X  -162.820, Y  +585.410, Z    +0.000, E1   -22.764, E3 +516955.604}
SPL {X  -162.820, Y  +587.676, Z    +0.000, E1   -22.853, E3 +516966.118}
SPL {X  -162.820, Y  +589.682, Z    +0.000, E1   -22.776, E3 +516976.648}
SPL {X  -162.820, Y  +591.720, Z    +0.000, E1   -22.868, E3 +516985.959}
SPL {X  -162.820, Y  +593.650, Z    +0.000, E1   -22.810, E3 +516996.029}
SPL {X  -162.820, Y  +595.830, Z    +0.000, E1   -22.828, E3 +517006.645}
SPL {X  -162.820, Y  +598.094, Z    +0.000, E1   -22.843, E3 +517017.758}
SPL {X  -162.820, Y  +600.420, Z    +0.000, E1   -22.826, E3 +517029.389}
SPL {X  -162.820, Y  +602.573, Z    +0.000, E1   -22.830, E3 +517039.974}
SPL {X  -162.820, Y  +604.828, Z    +0.000, E1   -22.784, E3 +517051.613}
SPL {X  -162.820, Y  +608.133, Z    +0.000, E1   -22.831, E3 +517067.730}
SPL {X  -162.820, Y  +611.103, Z    +0.000, E1   -22.785, E3 +517082.656}
SPL {X  -162.820, Y  +613.294, Z    +0.000, E1   -22.780, E3 +517093.529}
SPL {X  -162.820, Y  +615.356, Z    +0.000, E1   -22.799, E3 +517103.586}
SPL {X  -162.820, Y  +617.439, Z    +0.000, E1   -22.808, E3 +517113.845}
SPL {X  -162.820, Y  +619.665, Z    +0.000, E1   -22.817, E3 +517124.813}
SPL {X  -162.820, Y  +621.733, Z    +0.000, E1   -22.759, E3 +517135.537}
SPL {X  -162.820, Y  +624.076, Z    +0.000, E1   -22.774, E3 +517147.042}
SPL {X  -162.820, Y  +627.244, Z    +0.000, E1   -22.803, E3 +517162.724}
SPL {X  -162.820, Y  +630.349, Z    +0.000, E1   -22.766, E3 +517178.256}
SPL {X  -162.820, Y  +632.572, Z    +0.000, E1   -22.785, E3 +517189.063}
SPL {X  -162.820, Y  +634.507, Z    +0.000, E1   -22.784, E3 +517198.701}
SPL {X  -162.820, Y  +636.863, Z    +0.000, E1   -22.760, E3 +517210.624}
SPL {X  -162.820, Y  +640.111, Z    +0.000, E1   -22.809, E3 +517226.506}
SPL {X  -162.820, Y  +643.449, Z    +0.000, E1   -22.796, E3 +517243.024}
SPL {X  -162.820, Y  +645.630, Z    +0.000, E1   -22.795, E3 +517253.720}
SPL {X  -162.820, Y  +647.561, Z    +0.000, E1   -22.705, E3 +517264.171}
SPL {X  -162.820, Y  +651.051, Z    +0.000, E1   -22.833, E3 +517280.590}
SPL {X  -162.820, Y  +653.898, Z    +0.000, E1   -22.796, E3 +517294.776}
SPL {X  -162.820, Y  +656.161, Z    +0.000, E1   -22.812, E3 +517305.898}
SPL {X  -162.820, Y  +658.384, Z    +0.000, E1   -22.822, E3 +517316.764}
SPL {X  -162.820, Y  +660.215, Z    +0.000, E1   -22.649, E3 +517327.355}
SPL {X  -162.820, Y  +662.823, Z    +0.000, E1   -22.799, E3 +517339.062}
SPL {X  -162.820, Y  +665.112, Z    +0.000, E1   -22.835, E3 +517350.117}
SPL {X  -162.820, Y  +667.016, Z    +0.000, E1   -22.823, E3 +517359.545}
SPL {X  -162.820, Y  +668.960, Z    +0.000, E1   -22.773, E3 +517369.713}
SPL {X  -162.820, Y  +672.333, Z    +0.000, E1   -22.837, E3 +517386.049}
SPL {X  -162.812, Y  +675.071, Z    +0.000, E1   -22.742, E3 +517400.194}
SPL {X  -162.773, Y  +677.428, Z    +0.000, E1   -22.762, E3 +517411.791}
SPL {X  -162.691, Y  +679.987, Z    +0.000, E1   -22.794, E3 +517424.205}
SPL {X  -162.559, Y  +682.717, Z    +0.000, E1   -22.726, E3 +517438.388}
SPL {X  -162.349, Y  +685.880, Z    +0.000, E1   -22.738, E3 +517453.989}
SPL {X  -162.164, Y  +688.106, Z    +0.000, E1   -22.661, E3 +517465.510}
SPL {X  -161.938, Y  +690.422, Z    +0.000, E1   -22.769, E3 +517476.185}
SPL {X  -161.065, Y  +697.344, Z    +0.000, E1   -25.698, E3 +517485.304}
SPL {X  -158.553, Y  +710.529, Z    +0.000, E1   -30.890, E3 +517499.201}
ENDSPLINE

SPLINE
SPL {X  -161.215, Y  +696.305, Z    +0.000, E1   -20.575, E3 +517525.782}
SPL {X  -161.691, Y  +692.643, Z    +0.000, E1   -17.369, E3 +517541.970}
SPL {X  -162.534, Y  +683.153, Z    +0.000, E1   -10.475, E3 +517567.437}
SPL {X  -162.820, Y  +667.630, Z    +0.000, E1    -0.882, E3 +517561.414}
SPL {X  -162.820, Y  +661.883, Z    +0.000, E1    +3.373, E3 +517566.857}
SPL {X  -162.820, Y  +655.163, Z    +0.000, E1    +8.702, E3 +517566.455}
SPL {X  -162.820, Y  +634.515, Z    +0.000, E1   +26.439, E3 +517558.869}
ENDSPLINE

SPLINE
SPL {X  -162.820, Y  +638.080, Z    +0.000, E1   +18.858, E3 +517588.833}
ENDSPLINE

SPLINE
SPL {X  -162.820, Y  +623.278, Z    +0.000, E1   +28.723, E3 +517590.404}
SPL {X  -162.820, Y  +618.658, Z    +0.000, E1   +26.841, E3 +517619.013}
ENDSPLINE

SPLINE
SPL {X  -162.820, Y  +623.685, Z    +0.000, E1   +22.346, E3 +517631.319}
ENDSPLINE

